      Continuar_M353 : Bool;
      Entrar_M353 : Bool;
      EmiOK_M353 : Bool;
      FinLote_M354 : Bool;
      Especial_M354 : Bool;
      Bit_02_M354 : Bool;
      Retroceder_M354 : Bool;
      Retirar_M354 : Bool;
      Continuar_M354 : Bool;
      Entrar_M354 : Bool;
      EmiOK_M354 : Bool;
      FinLote_M355 : Bool;
      Especial_M355 : Bool;
      Bit_02_M355 : Bool;
      Retroceder_M355 : Bool;
      Retirar_M355 : Bool;
      Continuar_M355 : Bool;
      Entrar_M355 : Bool;
      EmiOK_M355 : Bool;
      FinLote_M356 : Bool;
      Especial_M356 : Bool;
      Bit_02_M356 : Bool;
      Retroceder_M356 : Bool;
      Retirar_M356 : Bool;
      Continuar_M356 : Bool;
      Entrar_M356 : Bool;
      EmiOK_M356 : Bool;
      FinLote_M357 : Bool;
      Especial_M357 : Bool;
      Bit_02_M357 : Bool;
      Retroceder_M357 : Bool;
      Retirar_M357 : Bool;
      Continuar_M357 : Bool;
      Entrar_M357 : Bool;
      EmiOK_M357 : Bool;
      FinLote_M358 : Bool;
      Especial_M358 : Bool;
      Bit_02_M358 : Bool;
      Retroceder_M358 : Bool;
      Retirar_M358 : Bool;
      Continuar_M358 : Bool;
      Entrar_M358 : Bool;
      EmiOK_M358 : Bool;
      FinLote_M359 : Bool;
      Especial_M359 : Bool;
      Bit_02_M359 : Bool;
      Retroceder_M359 : Bool;
      Retirar_M359 : Bool;
      Continuar_M359 : Bool;
      Entrar_M359 : Bool;
      EmiOK_M359 : Bool;
      FinLote_M360 : Bool;
      Especial_M360 : Bool;
      Bit_02_M360 : Bool;
      Retroceder_M360 : Bool;
      Retirar_M360 : Bool;
      Continuar_M360 : Bool;
      Entrar_M360 : Bool;
      EmiOK_M360 : Bool;
      FinLote_M361 : Bool;
      Especial_M361 : Bool;
      Bit_02_M361 : Bool;
      Retroceder_M361 : Bool;
      Retirar_M361 : Bool;
      Continuar_M361 : Bool;
      Entrar_M361 : Bool;
      EmiOK_M361 : Bool;
      FinLote_M362 : Bool;
      Especial_M362 : Bool;
      Bit_02_M362 : Bool;
      Retroceder_M362 : Bool;
      Retirar_M362 : Bool;
      Continuar_M362 : Bool;
      Entrar_M362 : Bool;
      EmiOK_M362 : Bool;
      FinLote_M363 : Bool;
      Especial_M363 : Bool;
      Bit_02_M363 : Bool;
      Retroceder_M363 : Bool;
      Retirar_M363 : Bool;
      Continuar_M363 : Bool;
      Entrar_M363 : Bool;
      EmiOK_M363 : Bool;
      FinLote_M364 : Bool;
      Especial_M364 : Bool;
      Bit_02_M364 : Bool;
      Retroceder_M364 : Bool;
      Retirar_M364 : Bool;
      Continuar_M364 : Bool;
      Entrar_M364 : Bool;
      EmiOK_M364 : Bool;
      FinLote_M365 : Bool;
      Especial_M365 : Bool;
      Bit_02_M365 : Bool;
      Retroceder_M365 : Bool;
      Retirar_M365 : Bool;
      Continuar_M365 : Bool;
      Entrar_M365 : Bool;
      EmiOK_M365 : Bool;
      FinLote_M366 : Bool;
      Especial_M366 : Bool;
      Bit_02_M366 : Bool;
      Retroceder_M366 : Bool;
      Retirar_M366 : Bool;
      Continuar_M366 : Bool;
      Entrar_M366 : Bool;
      EmiOK_M366 : Bool;
      FinLote_M367 : Bool;
      Especial_M367 : Bool;
      Bit_02_M367 : Bool;
      Retroceder_M367 : Bool;
      Retirar_M367 : Bool;
      Continuar_M367 : Bool;
      Entrar_M367 : Bool;
      EmiOK_M367 : Bool;
      FinLote_M368 : Bool;
      Especial_M368 : Bool;
      Bit_02_M368 : Bool;
      Retroceder_M368 : Bool;
      Retirar_M368 : Bool;
      Continuar_M368 : Bool;
      Entrar_M368 : Bool;
      EmiOK_M368 : Bool;
      FinLote_M369 : Bool;
      Especial_M369 : Bool;
      Bit_02_M369 : Bool;
      Retroceder_M369 : Bool;
      Retirar_M369 : Bool;
      Continuar_M369 : Bool;
      Entrar_M369 : Bool;
      EmiOK_M369 : Bool;
      FinLote_M370 : Bool;
      Especial_M370 : Bool;
      Bit_02_M370 : Bool;
      Retroceder_M370 : Bool;
      Retirar_M370 : Bool;
      Continuar_M370 : Bool;
      Entrar_M370 : Bool;
      EmiOK_M370 : Bool;
      FinLote_M371 : Bool;
      Especial_M371 : Bool;
      Bit_02_M371 : Bool;
      Retroceder_M371 : Bool;
      Retirar_M371 : Bool;
      Continuar_M371 : Bool;
      Entrar_M371 : Bool;
      EmiOK_M371 : Bool;
      FinLote_M372 : Bool;
      Especial_M372 : Bool;
      Bit_02_M372 : Bool;
      Retroceder_M372 : Bool;
      Retirar_M372 : Bool;
      Continuar_M372 : Bool;
      Entrar_M372 : Bool;
      EmiOK_M372 : Bool;
      FinLote_M373 : Bool;
      Especial_M373 : Bool;
      Bit_02_M373 : Bool;
      Retroceder_M373 : Bool;
      Retirar_M373 : Bool;
      Continuar_M373 : Bool;
      Entrar_M373 : Bool;
      EmiOK_M373 : Bool;
      FinLote_M374 : Bool;
      Especial_M374 : Bool;
      Bit_02_M374 : Bool;
      Retroceder_M374 : Bool;
      Retirar_M374 : Bool;
      Continuar_M374 : Bool;
      Entrar_M374 : Bool;
      EmiOK_M374 : Bool;
      FinLote_M375 : Bool;
      Especial_M375 : Bool;
      Bit_02_M375 : Bool;
      Retroceder_M375 : Bool;
      Retirar_M375 : Bool;
      Continuar_M375 : Bool;
      Entrar_M375 : Bool;
      EmiOK_M375 : Bool;
      FinLote_M376 : Bool;
      Especial_M376 : Bool;
      Bit_02_M376 : Bool;
      Retroceder_M376 : Bool;
      Retirar_M376 : Bool;
      Continuar_M376 : Bool;
      Entrar_M376 : Bool;
      EmiOK_M376 : Bool;
      FinLote_M377 : Bool;
      Especial_M377 : Bool;
      Bit_02_M377 : Bool;
      Retroceder_M377 : Bool;
      Retirar_M377 : Bool;
      Continuar_M377 : Bool;
      Entrar_M377 : Bool;
      EmiOK_M377 : Bool;
      FinLote_M378 : Bool;
      Especial_M378 : Bool;
      Bit_02_M378 : Bool;
      Retroceder_M378 : Bool;
      Retirar_M378 : Bool;
      Continuar_M378 : Bool;
      Entrar_M378 : Bool;
      EmiOK_M378 : Bool;
      FinLote_M379 : Bool;
      Especial_M379 : Bool;
      Bit_02_M379 : Bool;
      Retroceder_M379 : Bool;
      Retirar_M379 : Bool;
      Continuar_M379 : Bool;
      Entrar_M379 : Bool;
      EmiOK_M379 : Bool;
      FinLote_M380 : Bool;
      Especial_M380 : Bool;
      Bit_02_M380 : Bool;
      Retroceder_M380 : Bool;
      Retirar_M380 : Bool;
      Continuar_M380 : Bool;
      Entrar_M380 : Bool;
      EmiOK_M380 : Bool;
      FinLote_M381 : Bool;
      Especial_M381 : Bool;
      Bit_02_M381 : Bool;
      Retroceder_M381 : Bool;
      Retirar_M381 : Bool;
      Continuar_M381 : Bool;
      Entrar_M381 : Bool;
      EmiOK_M381 : Bool;
      FinLote_M382 : Bool;
      Especial_M382 : Bool;
      Bit_02_M382 : Bool;
      Retroceder_M382 : Bool;
      Retirar_M382 : Bool;
      Continuar_M382 : Bool;
      Entrar_M382 : Bool;
      EmiOK_M382 : Bool;
      FinLote_M383 : Bool;
      Especial_M383 : Bool;
      Bit_02_M383 : Bool;
      Retroceder_M383 : Bool;
      Retirar_M383 : Bool;
      Continuar_M383 : Bool;
      Entrar_M383 : Bool;
      EmiOK_M383 : Bool;
      FinLote_M384 : Bool;
      Especial_M384 : Bool;
      Bit_02_M384 : Bool;
      Retroceder_M384 : Bool;
      Retirar_M384 : Bool;
      Continuar_M384 : Bool;
      Entrar_M384 : Bool;
      EmiOK_M384 : Bool;
      FinLote_M385 : Bool;
      Especial_M385 : Bool;
      Bit_02_M385 : Bool;
      Retroceder_M385 : Bool;
      Retirar_M385 : Bool;
      Continuar_M385 : Bool;
      Entrar_M385 : Bool;
      EmiOK_M385 : Bool;
      FinLote_M386 : Bool;
      Especial_M386 : Bool;
      Bit_02_M386 : Bool;
      Retroceder_M386 : Bool;
      Retirar_M386 : Bool;
      Continuar_M386 : Bool;
      Entrar_M386 : Bool;
      EmiOK_M386 : Bool;
      FinLote_M387 : Bool;
      Especial_M387 : Bool;
      Bit_02_M387 : Bool;
      Retroceder_M387 : Bool;
      Retirar_M387 : Bool;
      Continuar_M387 : Bool;
      Entrar_M387 : Bool;
      EmiOK_M387 : Bool;
      FinLote_M388 : Bool;
      Especial_M388 : Bool;
      Bit_02_M388 : Bool;
      Retroceder_M388 : Bool;
      Retirar_M388 : Bool;
      Continuar_M388 : Bool;
      Entrar_M388 : Bool;
      EmiOK_M388 : Bool;
      FinLote_M389 : Bool;
      Especial_M389 : Bool;
      Bit_02_M389 : Bool;
      Retroceder_M389 : Bool;
      Retirar_M389 : Bool;
      Continuar_M389 : Bool;
      Entrar_M389 : Bool;
      EmiOK_M389 : Bool;
      FinLote_M390 : Bool;
      Especial_M390 : Bool;
      Bit_02_M390 : Bool;
      Retroceder_M390 : Bool;
      Retirar_M390 : Bool;
      Continuar_M390 : Bool;
      Entrar_M390 : Bool;
      EmiOK_M390 : Bool;
      FinLote_M391 : Bool;
      Especial_M391 : Bool;
      Bit_02_M391 : Bool;
      Retroceder_M391 : Bool;
      Retirar_M391 : Bool;
      Continuar_M391 : Bool;
      Entrar_M391 : Bool;
      EmiOK_M391 : Bool;
      FinLote_M392 : Bool;
      Especial_M392 : Bool;
      Bit_02_M392 : Bool;
      Retroceder_M392 : Bool;
      Retirar_M392 : Bool;
      Continuar_M392 : Bool;
      Entrar_M392 : Bool;
      EmiOK_M392 : Bool;
      FinLote_M393 : Bool;
      Especial_M393 : Bool;
      Bit_02_M393 : Bool;
      Retroceder_M393 : Bool;
      Retirar_M393 : Bool;
      Continuar_M393 : Bool;
      Entrar_M393 : Bool;
      EmiOK_M393 : Bool;
      FinLote_M394 : Bool;
      Especial_M394 : Bool;
      Bit_02_M394 : Bool;
      Retroceder_M394 : Bool;
      Retirar_M394 : Bool;
      Continuar_M394 : Bool;
      Entrar_M394 : Bool;
      EmiOK_M394 : Bool;
      FinLote_M395 : Bool;
      Especial_M395 : Bool;
      Bit_02_M395 : Bool;
      Retroceder_M395 : Bool;
      Retirar_M395 : Bool;
      Continuar_M395 : Bool;
      Entrar_M395 : Bool;
      EmiOK_M395 : Bool;
      FinLote_M396 : Bool;
      Especial_M396 : Bool;
      Bit_02_M396 : Bool;
      Retroceder_M396 : Bool;
      Retirar_M396 : Bool;
      Continuar_M396 : Bool;
      Entrar_M396 : Bool;
      EmiOK_M396 : Bool;
      FinLote_M397 : Bool;
      Especial_M397 : Bool;
      Bit_02_M397 : Bool;
      Retroceder_M397 : Bool;
      Retirar_M397 : Bool;
      Continuar_M397 : Bool;
      Entrar_M397 : Bool;
      EmiOK_M397 : Bool;
      FinLote_M398 : Bool;
      Especial_M398 : Bool;
      Bit_02_M398 : Bool;
      Retroceder_M398 : Bool;
      Retirar_M398 : Bool;
      Continuar_M398 : Bool;
      Entrar_M398 : Bool;
      EmiOK_M398 : Bool;
      FinLote_M399 : Bool;
      Especial_M399 : Bool;
      Bit_02_M399 : Bool;
      Retroceder_M399 : Bool;
      Retirar_M399 : Bool;
      Continuar_M399 : Bool;
      Entrar_M399 : Bool;
      EmiOK_M399 : Bool;
      FinLote_M400 : Bool;
      Especial_M400 : Bool;
      Bit_02_M400 : Bool;
      Retroceder_M400 : Bool;
      Retirar_M400 : Bool;
      Continuar_M400 : Bool;
      Entrar_M400 : Bool;
      EmiOK_M400 : Bool;
      FinLote_M401 : Bool;
      Especial_M401 : Bool;
      Bit_02_M401 : Bool;
      Retroceder_M401 : Bool;
      Retirar_M401 : Bool;
      Continuar_M401 : Bool;
      Entrar_M401 : Bool;
      EmiOK_M401 : Bool;
      FinLote_M402 : Bool;
      Especial_M402 : Bool;
      Bit_02_M402 : Bool;
      Retroceder_M402 : Bool;
      Retirar_M402 : Bool;
      Continuar_M402 : Bool;
      Entrar_M402 : Bool;
      EmiOK_M402 : Bool;
      FinLote_M403 : Bool;
      Especial_M403 : Bool;
      Bit_02_M403 : Bool;
      Retroceder_M403 : Bool;
      Retirar_M403 : Bool;
      Continuar_M403 : Bool;
      Entrar_M403 : Bool;
      EmiOK_M403 : Bool;
      FinLote_M404 : Bool;
      Especial_M404 : Bool;
      Bit_02_M404 : Bool;
      Retroceder_M404 : Bool;
      Retirar_M404 : Bool;
      Continuar_M404 : Bool;
      Entrar_M404 : Bool;
      EmiOK_M404 : Bool;
      FinLote_M405 : Bool;
      Especial_M405 : Bool;
      Bit_02_M405 : Bool;
      Retroceder_M405 : Bool;
      Retirar_M405 : Bool;
      Continuar_M405 : Bool;
      Entrar_M405 : Bool;
      EmiOK_M405 : Bool;
      FinLote_M406 : Bool;
      Especial_M406 : Bool;
      Bit_02_M406 : Bool;
      Retroceder_M406 : Bool;
      Retirar_M406 : Bool;
      Continuar_M406 : Bool;
      Entrar_M406 : Bool;
      EmiOK_M406 : Bool;
      FinLote_M407 : Bool;
      Especial_M407 : Bool;
      Bit_02_M407 : Bool;
      Retroceder_M407 : Bool;
      Retirar_M407 : Bool;
      Continuar_M407 : Bool;
      Entrar_M407 : Bool;
      EmiOK_M407 : Bool;
      FinLote_M408 : Bool;
      Especial_M408 : Bool;
      Bit_02_M408 : Bool;
      Retroceder_M408 : Bool;
      Retirar_M408 : Bool;
      Continuar_M408 : Bool;
      Entrar_M408 : Bool;
      EmiOK_M408 : Bool;
      FinLote_M409 : Bool;
      Especial_M409 : Bool;
      Bit_02_M409 : Bool;
      Retroceder_M409 : Bool;
      Retirar_M409 : Bool;
      Continuar_M409 : Bool;
      Entrar_M409 : Bool;
      EmiOK_M409 : Bool;
      FinLote_M410 : Bool;
      Especial_M410 : Bool;
      Bit_02_M410 : Bool;
      Retroceder_M410 : Bool;
      Retirar_M410 : Bool;
      Continuar_M410 : Bool;
      Entrar_M410 : Bool;
      EmiOK_M410 : Bool;
      FinLote_M411 : Bool;
      Especial_M411 : Bool;
      Bit_02_M411 : Bool;
      Retroceder_M411 : Bool;
      Retirar_M411 : Bool;
      Continuar_M411 : Bool;
      Entrar_M411 : Bool;
      EmiOK_M411 : Bool;
      FinLote_M412 : Bool;
      Especial_M412 : Bool;
      Bit_02_M412 : Bool;
      Retroceder_M412 : Bool;
      Retirar_M412 : Bool;
      Continuar_M412 : Bool;
      Entrar_M412 : Bool;
      EmiOK_M412 : Bool;
      FinLote_M413 : Bool;
      Especial_M413 : Bool;
      Bit_02_M413 : Bool;
      Retroceder_M413 : Bool;
      Retirar_M413 : Bool;
      Continuar_M413 : Bool;
      Entrar_M413 : Bool;
      EmiOK_M413 : Bool;
      FinLote_M414 : Bool;
      Especial_M414 : Bool;
      Bit_02_M414 : Bool;
      Retroceder_M414 : Bool;
      Retirar_M414 : Bool;
      Continuar_M414 : Bool;
      Entrar_M414 : Bool;
      EmiOK_M414 : Bool;
      FinLote_M415 : Bool;
      Especial_M415 : Bool;
      Bit_02_M415 : Bool;
      Retroceder_M415 : Bool;
      Retirar_M415 : Bool;
      Continuar_M415 : Bool;
      Entrar_M415 : Bool;
      EmiOK_M415 : Bool;
      FinLote_M416 : Bool;
      Especial_M416 : Bool;
      Bit_02_M416 : Bool;
      Retroceder_M416 : Bool;
      Retirar_M416 : Bool;
      Continuar_M416 : Bool;
      Entrar_M416 : Bool;
      EmiOK_M416 : Bool;
      FinLote_M417 : Bool;
      Especial_M417 : Bool;
      Bit_02_M417 : Bool;
      Retroceder_M417 : Bool;
      Retirar_M417 : Bool;
      Continuar_M417 : Bool;
      Entrar_M417 : Bool;
      EmiOK_M417 : Bool;
      FinLote_M418 : Bool;
      Especial_M418 : Bool;
      Bit_02_M418 : Bool;
      Retroceder_M418 : Bool;
      Retirar_M418 : Bool;
      Continuar_M418 : Bool;
      Entrar_M418 : Bool;
      EmiOK_M418 : Bool;
      FinLote_M419 : Bool;
      Especial_M419 : Bool;
      Bit_02_M419 : Bool;
      Retroceder_M419 : Bool;
      Retirar_M419 : Bool;
      Continuar_M419 : Bool;
      Entrar_M419 : Bool;
      EmiOK_M419 : Bool;
      FinLote_M420 : Bool;
      Especial_M420 : Bool;
      Bit_02_M420 : Bool;
      Retroceder_M420 : Bool;
      Retirar_M420 : Bool;
      Continuar_M420 : Bool;
      Entrar_M420 : Bool;
      EmiOK_M420 : Bool;
      FinLote_M421 : Bool;
      Especial_M421 : Bool;
      Bit_02_M421 : Bool;
      Retroceder_M421 : Bool;
      Retirar_M421 : Bool;
      Continuar_M421 : Bool;
      Entrar_M421 : Bool;
      EmiOK_M421 : Bool;
      FinLote_M422 : Bool;
      Especial_M422 : Bool;
      Bit_02_M422 : Bool;
      Retroceder_M422 : Bool;
      Retirar_M422 : Bool;
      Continuar_M422 : Bool;
      Entrar_M422 : Bool;
      EmiOK_M422 : Bool;
      FinLote_M423 : Bool;
      Especial_M423 : Bool;
      Bit_02_M423 : Bool;
      Retroceder_M423 : Bool;
      Retirar_M423 : Bool;
      Continuar_M423 : Bool;
      Entrar_M423 : Bool;
      EmiOK_M423 : Bool;
      FinLote_M424 : Bool;
      Especial_M424 : Bool;
      Bit_02_M424 : Bool;
      Retroceder_M424 : Bool;
      Retirar_M424 : Bool;
      Continuar_M424 : Bool;
      Entrar_M424 : Bool;
      EmiOK_M424 : Bool;
      FinLote_M425 : Bool;
      Especial_M425 : Bool;
      Bit_02_M425 : Bool;
      Retroceder_M425 : Bool;
      Retirar_M425 : Bool;
      Continuar_M425 : Bool;
      Entrar_M425 : Bool;
      EmiOK_M425 : Bool;
      FinLote_M426 : Bool;
      Especial_M426 : Bool;
      Bit_02_M426 : Bool;
      Retroceder_M426 : Bool;
      Retirar_M426 : Bool;
      Continuar_M426 : Bool;
      Entrar_M426 : Bool;
      EmiOK_M426 : Bool;
      FinLote_M427 : Bool;
      Especial_M427 : Bool;
      Bit_02_M427 : Bool;
      Retroceder_M427 : Bool;
      Retirar_M427 : Bool;
      Continuar_M427 : Bool;
      Entrar_M427 : Bool;
      EmiOK_M427 : Bool;
      FinLote_M428 : Bool;
      Especial_M428 : Bool;
      Bit_02_M428 : Bool;
      Retroceder_M428 : Bool;
      Retirar_M428 : Bool;
      Continuar_M428 : Bool;
      Entrar_M428 : Bool;
      EmiOK_M428 : Bool;
      FinLote_M429 : Bool;
      Especial_M429 : Bool;
      Bit_02_M429 : Bool;
      Retroceder_M429 : Bool;
      Retirar_M429 : Bool;
      Continuar_M429 : Bool;
      Entrar_M429 : Bool;
      EmiOK_M429 : Bool;
      FinLote_M430 : Bool;
      Especial_M430 : Bool;
      Bit_02_M430 : Bool;
      Retroceder_M430 : Bool;
      Retirar_M430 : Bool;
      Continuar_M430 : Bool;
      Entrar_M430 : Bool;
      EmiOK_M430 : Bool;
      FinLote_M431 : Bool;
      Especial_M431 : Bool;
      Bit_02_M431 : Bool;
      Retroceder_M431 : Bool;
      Retirar_M431 : Bool;
      Continuar_M431 : Bool;
      Entrar_M431 : Bool;
      EmiOK_M431 : Bool;
      FinLote_M432 : Bool;
      Especial_M432 : Bool;
      Bit_02_M432 : Bool;
      Retroceder_M432 : Bool;
      Retirar_M432 : Bool;
      Continuar_M432 : Bool;
      Entrar_M432 : Bool;
      EmiOK_M432 : Bool;
      FinLote_M433 : Bool;
      Especial_M433 : Bool;
      Bit_02_M433 : Bool;
      Retroceder_M433 : Bool;
      Retirar_M433 : Bool;
      Continuar_M433 : Bool;
      Entrar_M433 : Bool;
      EmiOK_M433 : Bool;
      FinLote_M434 : Bool;
      Especial_M434 : Bool;
      Bit_02_M434 : Bool;
      Retroceder_M434 : Bool;
      Retirar_M434 : Bool;
      Continuar_M434 : Bool;
      Entrar_M434 : Bool;
      EmiOK_M434 : Bool;
      FinLote_M435 : Bool;
      Especial_M435 : Bool;
      Bit_02_M435 : Bool;
      Retroceder_M435 : Bool;
      Retirar_M435 : Bool;
      Continuar_M435 : Bool;
      Entrar_M435 : Bool;
      EmiOK_M435 : Bool;
      FinLote_M436 : Bool;
      Especial_M436 : Bool;
      Bit_02_M436 : Bool;
      Retroceder_M436 : Bool;
      Retirar_M436 : Bool;
      Continuar_M436 : Bool;
      Entrar_M436 : Bool;
      EmiOK_M436 : Bool;
      FinLote_M437 : Bool;
      Especial_M437 : Bool;
      Bit_02_M437 : Bool;
      Retroceder_M437 : Bool;
      Retirar_M437 : Bool;
      Continuar_M437 : Bool;
      Entrar_M437 : Bool;
      EmiOK_M437 : Bool;
      FinLote_M438 : Bool;
      Especial_M438 : Bool;
      Bit_02_M438 : Bool;
      Retroceder_M438 : Bool;
      Retirar_M438 : Bool;
      Continuar_M438 : Bool;
      Entrar_M438 : Bool;
      EmiOK_M438 : Bool;
      FinLote_M439 : Bool;
      Especial_M439 : Bool;
      Bit_02_M439 : Bool;
      Retroceder_M439 : Bool;
      Retirar_M439 : Bool;
      Continuar_M439 : Bool;
      Entrar_M439 : Bool;
      EmiOK_M439 : Bool;
      FinLote_M440 : Bool;
      Especial_M440 : Bool;
      Bit_02_M440 : Bool;
      Retroceder_M440 : Bool;
      Retirar_M440 : Bool;
      Continuar_M440 : Bool;
      Entrar_M440 : Bool;
      EmiOK_M440 : Bool;
      FinLote_M441 : Bool;
      Especial_M441 : Bool;
      Bit_02_M441 : Bool;
      Retroceder_M441 : Bool;
      Retirar_M441 : Bool;
      Continuar_M441 : Bool;
      Entrar_M441 : Bool;
      EmiOK_M441 : Bool;
      FinLote_M442 : Bool;
      Especial_M442 : Bool;
      Bit_02_M442 : Bool;
      Retroceder_M442 : Bool;
      Retirar_M442 : Bool;
      Continuar_M442 : Bool;
      Entrar_M442 : Bool;
      EmiOK_M442 : Bool;
      FinLote_M443 : Bool;
      Especial_M443 : Bool;
      Bit_02_M443 : Bool;
      Retroceder_M443 : Bool;
      Retirar_M443 : Bool;
      Continuar_M443 : Bool;
      Entrar_M443 : Bool;
      EmiOK_M443 : Bool;
      FinLote_M444 : Bool;
      Especial_M444 : Bool;
      Bit_02_M444 : Bool;
      Retroceder_M444 : Bool;
      Retirar_M444 : Bool;
      Continuar_M444 : Bool;
      Entrar_M444 : Bool;
      EmiOK_M444 : Bool;
      FinLote_M445 : Bool;
      Especial_M445 : Bool;
      Bit_02_M445 : Bool;
      Retroceder_M445 : Bool;
      Retirar_M445 : Bool;
      Continuar_M445 : Bool;
      Entrar_M445 : Bool;
      EmiOK_M445 : Bool;
      FinLote_M446 : Bool;
      Especial_M446 : Bool;
      Bit_02_M446 : Bool;
      Retroceder_M446 : Bool;
      Retirar_M446 : Bool;
      Continuar_M446 : Bool;
      Entrar_M446 : Bool;
      EmiOK_M446 : Bool;
      FinLote_M447 : Bool;
      Especial_M447 : Bool;
      Bit_02_M447 : Bool;
      Retroceder_M447 : Bool;
      Retirar_M447 : Bool;
      Continuar_M447 : Bool;
      Entrar_M447 : Bool;
      EmiOK_M447 : Bool;
      FinLote_M448 : Bool;
      Especial_M448 : Bool;
      Bit_02_M448 : Bool;
      Retroceder_M448 : Bool;
      Retirar_M448 : Bool;
      Continuar_M448 : Bool;
      Entrar_M448 : Bool;
      EmiOK_M448 : Bool;
      FinLote_M449 : Bool;
      Especial_M449 : Bool;
      Bit_02_M449 : Bool;
      Retroceder_M449 : Bool;
      Retirar_M449 : Bool;
      Continuar_M449 : Bool;
      Entrar_M449 : Bool;
      EmiOK_M449 : Bool;
      FinLote_M450 : Bool;
      Especial_M450 : Bool;
      Bit_02_M450 : Bool;
      Retroceder_M450 : Bool;
      Retirar_M450 : Bool;
      Continuar_M450 : Bool;
      Entrar_M450 : Bool;
      EmiOK_M450 : Bool;
      FinLote_M451 : Bool;
      Especial_M451 : Bool;
      Bit_02_M451 : Bool;
      Retroceder_M451 : Bool;
      Retirar_M451 : Bool;
      Continuar_M451 : Bool;
      Entrar_M451 : Bool;
      EmiOK_M451 : Bool;
      FinLote_M452 : Bool;
      Especial_M452 : Bool;
      Bit_02_M452 : Bool;
      Retroceder_M452 : Bool;
      Retirar_M452 : Bool;
      Continuar_M452 : Bool;
      Entrar_M452 : Bool;
      EmiOK_M452 : Bool;
      FinLote_M453 : Bool;
      Especial_M453 : Bool;
      Bit_02_M453 : Bool;
      Retroceder_M453 : Bool;
      Retirar_M453 : Bool;
      Continuar_M453 : Bool;
      Entrar_M453 : Bool;
      EmiOK_M453 : Bool;
      FinLote_M454 : Bool;
      Especial_M454 : Bool;
      Bit_02_M454 : Bool;
      Retroceder_M454 : Bool;
      Retirar_M454 : Bool;
      Continuar_M454 : Bool;
      Entrar_M454 : Bool;
      EmiOK_M454 : Bool;
      FinLote_M455 : Bool;
      Especial_M455 : Bool;
      Bit_02_M455 : Bool;
      Retroceder_M455 : Bool;
      Retirar_M455 : Bool;
      Continuar_M455 : Bool;
      Entrar_M455 : Bool;
      EmiOK_M455 : Bool;
      FinLote_M456 : Bool;
      Especial_M456 : Bool;
      Bit_02_M456 : Bool;
      Retroceder_M456 : Bool;
      Retirar_M456 : Bool;
      Continuar_M456 : Bool;
      Entrar_M456 : Bool;
      EmiOK_M456 : Bool;
      FinLote_M457 : Bool;
      Especial_M457 : Bool;
      Bit_02_M457 : Bool;
      Retroceder_M457 : Bool;
      Retirar_M457 : Bool;
      Continuar_M457 : Bool;
      Entrar_M457 : Bool;
      EmiOK_M457 : Bool;
      FinLote_M458 : Bool;
      Especial_M458 : Bool;
      Bit_02_M458 : Bool;
      Retroceder_M458 : Bool;
      Retirar_M458 : Bool;
      Continuar_M458 : Bool;
      Entrar_M458 : Bool;
      EmiOK_M458 : Bool;
      FinLote_M459 : Bool;
      Especial_M459 : Bool;
      Bit_02_M459 : Bool;
      Retroceder_M459 : Bool;
      Retirar_M459 : Bool;
      Continuar_M459 : Bool;
      Entrar_M459 : Bool;
      EmiOK_M459 : Bool;
      FinLote_M460 : Bool;
      Especial_M460 : Bool;
      Bit_02_M460 : Bool;
      Retroceder_M460 : Bool;
      Retirar_M460 : Bool;
      Continuar_M460 : Bool;
      Entrar_M460 : Bool;
      EmiOK_M460 : Bool;
      FinLote_M461 : Bool;
      Especial_M461 : Bool;
      Bit_02_M461 : Bool;
      Retroceder_M461 : Bool;
      Retirar_M461 : Bool;
      Continuar_M461 : Bool;
      Entrar_M461 : Bool;
      EmiOK_M461 : Bool;
      FinLote_M462 : Bool;
      Especial_M462 : Bool;
      Bit_02_M462 : Bool;
      Retroceder_M462 : Bool;
      Retirar_M462 : Bool;
      Continuar_M462 : Bool;
      Entrar_M462 : Bool;
      EmiOK_M462 : Bool;
      FinLote_M463 : Bool;
      Especial_M463 : Bool;
      Bit_02_M463 : Bool;
      Retroceder_M463 : Bool;
      Retirar_M463 : Bool;
      Continuar_M463 : Bool;
      Entrar_M463 : Bool;
      EmiOK_M463 : Bool;
      FinLote_M464 : Bool;
      Especial_M464 : Bool;
      Bit_02_M464 : Bool;
      Retroceder_M464 : Bool;
      Retirar_M464 : Bool;
      Continuar_M464 : Bool;
      Entrar_M464 : Bool;
      EmiOK_M464 : Bool;
      FinLote_M465 : Bool;
      Especial_M465 : Bool;
      Bit_02_M465 : Bool;
      Retroceder_M465 : Bool;
      Retirar_M465 : Bool;
      Continuar_M465 : Bool;
      Entrar_M465 : Bool;
      EmiOK_M465 : Bool;
      FinLote_M466 : Bool;
      Especial_M466 : Bool;
      Bit_02_M466 : Bool;
      Retroceder_M466 : Bool;
      Retirar_M466 : Bool;
      Continuar_M466 : Bool;
      Entrar_M466 : Bool;
      EmiOK_M466 : Bool;
      FinLote_M467 : Bool;
      Especial_M467 : Bool;
      Bit_02_M467 : Bool;
      Retroceder_M467 : Bool;
      Retirar_M467 : Bool;
      Continuar_M467 : Bool;
      Entrar_M467 : Bool;
      EmiOK_M467 : Bool;
      FinLote_M468 : Bool;
      Especial_M468 : Bool;
      Bit_02_M468 : Bool;
      Retroceder_M468 : Bool;
      Retirar_M468 : Bool;
      Continuar_M468 : Bool;
      Entrar_M468 : Bool;
      EmiOK_M468 : Bool;
      FinLote_M469 : Bool;
      Especial_M469 : Bool;
      Bit_02_M469 : Bool;
      Retroceder_M469 : Bool;
      Retirar_M469 : Bool;
      Continuar_M469 : Bool;
      Entrar_M469 : Bool;
      EmiOK_M469 : Bool;
      FinLote_M470 : Bool;
      Especial_M470 : Bool;
      Bit_02_M470 : Bool;
      Retroceder_M470 : Bool;
      Retirar_M470 : Bool;
      Continuar_M470 : Bool;
      Entrar_M470 : Bool;
      EmiOK_M470 : Bool;
      FinLote_M471 : Bool;
      Especial_M471 : Bool;
      Bit_02_M471 : Bool;
      Retroceder_M471 : Bool;
      Retirar_M471 : Bool;
      Continuar_M471 : Bool;
      Entrar_M471 : Bool;
      EmiOK_M471 : Bool;
      FinLote_M472 : Bool;
      Especial_M472 : Bool;
      Bit_02_M472 : Bool;
      Retroceder_M472 : Bool;
      Retirar_M472 : Bool;
      Continuar_M472 : Bool;
      Entrar_M472 : Bool;
      EmiOK_M472 : Bool;
      FinLote_M473 : Bool;
      Especial_M473 : Bool;
      Bit_02_M473 : Bool;
      Retroceder_M473 : Bool;
      Retirar_M473 : Bool;
      Continuar_M473 : Bool;
      Entrar_M473 : Bool;
      EmiOK_M473 : Bool;
      FinLote_M474 : Bool;
      Especial_M474 : Bool;
      Bit_02_M474 : Bool;
      Retroceder_M474 : Bool;
      Retirar_M474 : Bool;
      Continuar_M474 : Bool;
      Entrar_M474 : Bool;
      EmiOK_M474 : Bool;
      FinLote_M475 : Bool;
      Especial_M475 : Bool;
      Bit_02_M475 : Bool;
      Retroceder_M475 : Bool;
      Retirar_M475 : Bool;
      Continuar_M475 : Bool;
      Entrar_M475 : Bool;
      EmiOK_M475 : Bool;
      FinLote_M476 : Bool;
      Especial_M476 : Bool;
      Bit_02_M476 : Bool;
      Retroceder_M476 : Bool;
      Retirar_M476 : Bool;
      Continuar_M476 : Bool;
      Entrar_M476 : Bool;
      EmiOK_M476 : Bool;
      FinLote_M477 : Bool;
      Especial_M477 : Bool;
      Bit_02_M477 : Bool;
      Retroceder_M477 : Bool;
      Retirar_M477 : Bool;
      Continuar_M477 : Bool;
      Entrar_M477 : Bool;
      EmiOK_M477 : Bool;
      FinLote_M478 : Bool;
      Especial_M478 : Bool;
      Bit_02_M478 : Bool;
      Retroceder_M478 : Bool;
      Retirar_M478 : Bool;
      Continuar_M478 : Bool;
      Entrar_M478 : Bool;
      EmiOK_M478 : Bool;
      FinLote_M479 : Bool;
      Especial_M479 : Bool;
      Bit_02_M479 : Bool;
      Retroceder_M479 : Bool;
      Retirar_M479 : Bool;
      Continuar_M479 : Bool;
      Entrar_M479 : Bool;
      EmiOK_M479 : Bool;
      FinLote_M480 : Bool;
      Especial_M480 : Bool;
      Bit_02_M480 : Bool;
      Retroceder_M480 : Bool;
      Retirar_M480 : Bool;
      Continuar_M480 : Bool;
      Entrar_M480 : Bool;
      EmiOK_M480 : Bool;
      FinLote_M481 : Bool;
      Especial_M481 : Bool;
      Bit_02_M481 : Bool;
      Retroceder_M481 : Bool;
      Retirar_M481 : Bool;
      Continuar_M481 : Bool;
      Entrar_M481 : Bool;
      EmiOK_M481 : Bool;
      FinLote_M482 : Bool;
      Especial_M482 : Bool;
      Bit_02_M482 : Bool;
      Retroceder_M482 : Bool;
      Retirar_M482 : Bool;
      Continuar_M482 : Bool;
      Entrar_M482 : Bool;
      EmiOK_M482 : Bool;
      FinLote_M483 : Bool;
      Especial_M483 : Bool;
      Bit_02_M483 : Bool;
      Retroceder_M483 : Bool;
      Retirar_M483 : Bool;
      Continuar_M483 : Bool;
      Entrar_M483 : Bool;
      EmiOK_M483 : Bool;
      FinLote_M484 : Bool;
      Especial_M484 : Bool;
      Bit_02_M484 : Bool;
      Retroceder_M484 : Bool;
      Retirar_M484 : Bool;
      Continuar_M484 : Bool;
      Entrar_M484 : Bool;
      EmiOK_M484 : Bool;
      FinLote_M485 : Bool;
      Especial_M485 : Bool;
      Bit_02_M485 : Bool;
      Retroceder_M485 : Bool;
      Retirar_M485 : Bool;
      Continuar_M485 : Bool;
      Entrar_M485 : Bool;
      EmiOK_M485 : Bool;
      FinLote_M486 : Bool;
      Especial_M486 : Bool;
      Bit_02_M486 : Bool;
      Retroceder_M486 : Bool;
      Retirar_M486 : Bool;
      Continuar_M486 : Bool;
      Entrar_M486 : Bool;
      EmiOK_M486 : Bool;
      FinLote_M487 : Bool;
      Especial_M487 : Bool;
      Bit_02_M487 : Bool;
      Retroceder_M487 : Bool;
      Retirar_M487 : Bool;
      Continuar_M487 : Bool;
      Entrar_M487 : Bool;
      EmiOK_M487 : Bool;
      FinLote_M488 : Bool;
      Especial_M488 : Bool;
      Bit_02_M488 : Bool;
      Retroceder_M488 : Bool;
      Retirar_M488 : Bool;
      Continuar_M488 : Bool;
      Entrar_M488 : Bool;
      EmiOK_M488 : Bool;
      FinLote_M489 : Bool;
      Especial_M489 : Bool;
      Bit_02_M489 : Bool;
      Retroceder_M489 : Bool;
      Retirar_M489 : Bool;
      Continuar_M489 : Bool;
      Entrar_M489 : Bool;
      EmiOK_M489 : Bool;
      FinLote_M490 : Bool;
      Especial_M490 : Bool;
      Bit_02_M490 : Bool;
      Retroceder_M490 : Bool;
      Retirar_M490 : Bool;
      Continuar_M490 : Bool;
      Entrar_M490 : Bool;
      EmiOK_M490 : Bool;
      FinLote_M491 : Bool;
      Especial_M491 : Bool;
      Bit_02_M491 : Bool;
      Retroceder_M491 : Bool;
      Retirar_M491 : Bool;
      Continuar_M491 : Bool;
      Entrar_M491 : Bool;
      EmiOK_M491 : Bool;
      FinLote_M492 : Bool;
      Especial_M492 : Bool;
      Bit_02_M492 : Bool;
      Retroceder_M492 : Bool;
      Retirar_M492 : Bool;
      Continuar_M492 : Bool;
      Entrar_M492 : Bool;
      EmiOK_M492 : Bool;
      FinLote_M493 : Bool;
      Especial_M493 : Bool;
      Bit_02_M493 : Bool;
      Retroceder_M493 : Bool;
      Retirar_M493 : Bool;
      Continuar_M493 : Bool;
      Entrar_M493 : Bool;
      EmiOK_M493 : Bool;
      FinLote_M494 : Bool;
      Especial_M494 : Bool;
      Bit_02_M494 : Bool;
      Retroceder_M494 : Bool;
      Retirar_M494 : Bool;
      Continuar_M494 : Bool;
      Entrar_M494 : Bool;
      EmiOK_M494 : Bool;
      FinLote_M495 : Bool;
      Especial_M495 : Bool;
      Bit_02_M495 : Bool;
      Retroceder_M495 : Bool;
      Retirar_M495 : Bool;
      Continuar_M495 : Bool;
      Entrar_M495 : Bool;
      EmiOK_M495 : Bool;
      FinLote_M496 : Bool;
      Especial_M496 : Bool;
      Bit_02_M496 : Bool;
      Retroceder_M496 : Bool;
      Retirar_M496 : Bool;
      Continuar_M496 : Bool;
      Entrar_M496 : Bool;
      EmiOK_M496 : Bool;
      FinLote_M497 : Bool;
      Especial_M497 : Bool;
      Bit_02_M497 : Bool;
      Retroceder_M497 : Bool;
      Retirar_M497 : Bool;
      Continuar_M497 : Bool;
      Entrar_M497 : Bool;
      EmiOK_M497 : Bool;
      FinLote_M498 : Bool;
      Especial_M498 : Bool;
      Bit_02_M498 : Bool;
      Retroceder_M498 : Bool;
      Retirar_M498 : Bool;
      Continuar_M498 : Bool;
      Entrar_M498 : Bool;
      EmiOK_M498 : Bool;
      FinLote_M499 : Bool;
      Especial_M499 : Bool;
      Bit_02_M499 : Bool;
      Retroceder_M499 : Bool;
      Retirar_M499 : Bool;
      Continuar_M499 : Bool;
      Entrar_M499 : Bool;
      EmiOK_M499 : Bool;
      FinLote_M500 : Bool;
      Especial_M500 : Bool;
      Bit_02_M500 : Bool;
      Retroceder_M500 : Bool;
      Retirar_M500 : Bool;
      Continuar_M500 : Bool;
      Entrar_M500 : Bool;
      EmiOK_M500 : Bool;
      Bit_00_CCPIF : Bool;
      Bit_01_CCPIF : Bool;
      Rearme_CCPIF : Bool;
      Bit_03_CCPIF : Bool;
      Reset_CCPIF : Bool;
      Paro_CCPIF : Bool;
      Marcha_CCPIF : Bool;
      EmiOK_CCPIF : Bool;
      Bit_00_CBOX1 : Bool;
      Bit_01_CBOX1 : Bool;
      Rearme_CBOX1 : Bool;
      Bit_03_CBOX1 : Bool;
      Reset_CBOX1 : Bool;
      Paro_CBOX1 : Bool;
      Marcha_CBOX1 : Bool;
      EmiOK_CBOX1 : Bool;
      Bit_00_CBOX2 : Bool;
      Bit_01_CBOX2 : Bool;
      Rearme_CBOX2 : Bool;
      Bit_03_CBOX2 : Bool;
      Reset_CBOX2 : Bool;
      Paro_CBOX2 : Bool;
      Marcha_CBOX2 : Bool;
      EmiOK_CBOX2 : Bool;
      Bit_00_CBOX3 : Bool;
      Bit_01_CBOX3 : Bool;
      Rearme_CBOX3 : Bool;
      Bit_03_CBOX3 : Bool;
      Reset_CBOX3 : Bool;
      Paro_CBOX3 : Bool;
      Marcha_CBOX3 : Bool;
      EmiOK_CBOX3 : Bool;
      Bit_00_CBOX4 : Bool;
      Bit_01_CBOX4 : Bool;
      Rearme_CBOX4 : Bool;
      Bit_03_CBOX4 : Bool;
      Reset_CBOX4 : Bool;
      Paro_CBOX4 : Bool;
      Marcha_CBOX4 : Bool;
      EmiOK_CBOX4 : Bool;
      Bit_00_CBOX5 : Bool;
      Bit_01_CBOX5 : Bool;
      Rearme_CBOX5 : Bool;
      Bit_03_CBOX5 : Bool;
      Reset_CBOX5 : Bool;
      Paro_CBOX5 : Bool;
      Marcha_CBOX5 : Bool;
      EmiOK_CBOX5 : Bool;
      Bit_00_CBOX6 : Bool;
      Bit_01_CBOX6 : Bool;
      Rearme_CBOX6 : Bool;
      Bit_03_CBOX6 : Bool;
      Reset_CBOX6 : Bool;
      Paro_CBOX6 : Bool;
      Marcha_CBOX6 : Bool;
      EmiOK_CBOX6 : Bool;
      Bit_00_CBOX7 : Bool;
      Bit_01_CBOX7 : Bool;
      Rearme_CBOX7 : Bool;
      Bit_03_CBOX7 : Bool;
      Reset_CBOX7 : Bool;
      Paro_CBOX7 : Bool;
      Marcha_CBOX7 : Bool;
      EmiOK_CBOX7 : Bool;
      Bit_00_CBOX8 : Bool;
      Bit_01_CBOX8 : Bool;
      Rearme_CBOX8 : Bool;
      Bit_03_CBOX8 : Bool;
      Reset_CBOX8 : Bool;
      Paro_CBOX8 : Bool;
      Marcha_CBOX8 : Bool;
      EmiOK_CBOX8 : Bool;
      Bit_00_CBOX9 : Bool;
      Bit_01_CBOX9 : Bool;
      Rearme_CBOX9 : Bool;
      Bit_03_CBOX9 : Bool;
      Reset_CBOX9 : Bool;
      Paro_CBOX9 : Bool;
      Marcha_CBOX9 : Bool;
      EmiOK_CBOX9 : Bool;
      Especial : Array[1..128] of Word;
   END_VAR
BEGIN
END_DATA_BLOCK

DATA_BLOCK "DB601_PeinesQuimarox"   // DB601
{ S7_Optimized_Access := 'FALSE' }
AUTHOR : Naibes
// stored: AutoNumber false
   VAR RETAIN
      Quimarox : Array[1.."CTE_MaxNumQuimarox"] of Struct
         vagon { S7_SetPoint := 'True'} : Array[1.."CTE_MaxNumVagones"] of "CBS_Carrier";
      END_STRUCT;
   END_VAR
BEGIN
END_DATA_BLOCK

DATA_BLOCK "DB602_ElementosQuimarox"   // DB602
{ S7_Optimized_Access := 'FALSE' }
// stored: AutoNumber false
   VAR RETAIN
      Quimarox : Array[1.."CTE_MaxNumQuimarox"] of Struct
         Elementos { S7_SetPoint := 'True'} : Array[1.."CTE_MaxNumElementos"] of "CBS_Elemento";
      END_STRUCT;
   END_VAR
BEGIN
   Quimarox[1].Elementos[1].posicion_real_elemento := 700.0;
   Quimarox[1].Elementos[2].posicion_real_elemento := 7700.0;
   Quimarox[1].Elementos[3].posicion_real_elemento := 14890.0;
   Quimarox[1].Elementos[4].posicion_real_elemento := 18000.0;
   Quimarox[1].Elementos[5].posicion_real_elemento := 6870.7;
   Quimarox[1].Elementos[1..5].ventana_minima := 50;
   Quimarox[1].Elementos[1].ventana_maxima := 1400;
   Quimarox[1].Elementos[2..5].ventana_maxima := 1550;
   Quimarox[1].Elementos[6..50].Numero_carrier := 11;
   Quimarox[1].Elementos[6..34].Avance_carrier := 1069;
   Quimarox[1].Elementos[35..47].Avance_carrier := 1079;
   Quimarox[1].Elementos[48..50].Avance_carrier := 1083;
END_DATA_BLOCK

DATA_BLOCK "DB1903_ASI_DIAG"   // DB1903
{ S7_Optimized_Access := 'FALSE'; DB_Accessible_From_OPC_UA := 'FALSE' }
// stored: AutoNumber false, DBAccessibleFromOPCUA false
   VAR
      ASI_Gateway_Error : Bool;
      IP_GW { S7_SetPoint := 'True'} : Array[1..16] of "ASI_GW_DATOS";
      ASI3_GW_C1 : Array[1..16] of "ASI3_Diag_GW";
      ASI3_GW_C2 : Array[1..16] of "ASI3_Diag_GW";
      ASI5_GW_Flags { S7_SetPoint := 'True'} : Array[1..16] of "ASI5_Flags";
      ASI5_GW_C1 : Array[1..16] of "ASI5_Diag_GW";
      ASI5_GW_C2 : Array[1..16] of "ASI5_Diag_GW";
   END_VAR
BEGIN
END_DATA_BLOCK

ORGANIZATION_BLOCK "OB1_Principal"   // OB1, LAD, ProgramCycle
TITLE = "Main Program Sweep (Cycle)"
{ S7_Optimized_Access := 'FALSE' }
AUTHOR : ESTANDAR
NAME : 20150525
VERSION : 3.1
// stored: AutoNumber false, SetENOAutomatically false
   VAR_TEMP
      OB1_EV_CLASS : Byte;   // Bits 0-3 = 1 (Coming event), Bits 4-7 = 1 (Event class 1)
      OB1_SCAN_1 : Byte;   // 1 (Cold restart scan 1 of OB 1), 3 (Scan 2-n of OB 1)
      OB1_PRIORITY : Byte;   // Priority of OB Execution
      OB1_OB_NUMBR : Byte;   // 1 (Organization block 1, OB1)
      OB1_RESERVED_1 : Byte;   // Reserved for system
      OB1_RESERVED_2 : Byte;   // Reserved for system
      OB1_PREV_CYCLE : Int;   // Cycle time of previous OB1 scan (milliseconds)
      OB1_MIN_CYCLE : Int;   // Minimum cycle time of OB1 (milliseconds)
      OB1_MAX_CYCLE : Int;   // Maximum cycle time of OB1 (milliseconds)
      OB1_DATE_TIME : Date_And_Time;   // Date and time OB1 started
      indice : UInt;
   END_VAR
   VAR_TEMP   // added for the SCL form of the ladder/FBD networks
      _w1 : Bool;
   END_VAR
BEGIN

REGION Network 1: Marcas Auxiliares CCPIF
   // *******************************************************************
   // * FUNCION: Generación marcas Auxiliares Generales del sistema     *
   // *******************************************************************
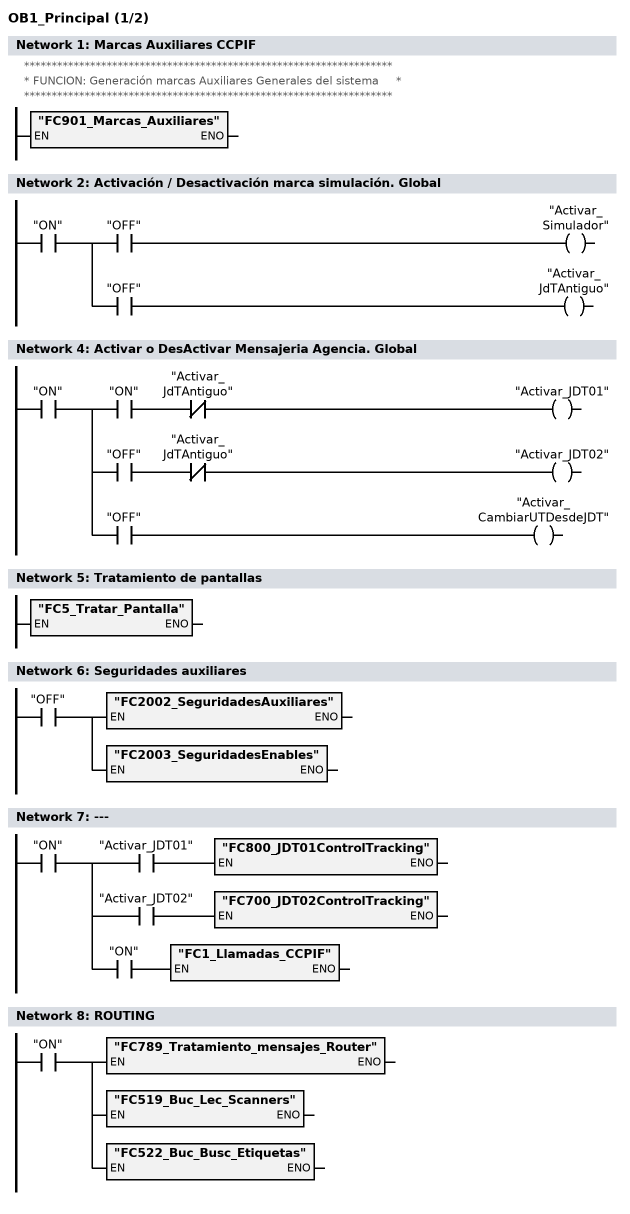
   RUNG wire#powerrail
      "FC901_Marcas_Auxiliares"()
   END_RUNG
   // the same network as SCL:
   "FC901_Marcas_Auxiliares"();
END_REGION

REGION Network 2: Activación / Desactivación marca simulación. Global
   RUNG wire#powerrail
      Contact( "ON" )
      wire#w1
      Contact( "OFF" )
      Coil( "Activar_Simulador" )
   END_RUNG
   RUNG wire#w1
      Contact( "OFF" )
      Coil( "Activar_JdTAntiguo" )
   END_RUNG
   // the same network as SCL:
   "Activar_Simulador" := "ON" AND "OFF";
   "Activar_JdTAntiguo" := "ON" AND "OFF";
END_REGION

NETWORK
TITLE = Cuando se desactive el JDT antiguo, tenemos que borrarnos todas las ordenes que se pudiesen quedar activas
// de lo contrario, habria problemas al realizar el cambio. Pablo
////////////////////////////////////////////////////////////////////////
////////////////////////////////////////////////////////////////////////
////////////////////////////////////////////////////////////////////////
/// --- Control de Cambio de Modo
      SET;
      A     "Activar_JdTAntiguo";
      FN    "Memo_JdTAntiguo_Desactivado";
      JC    BorradoDatos_CambioModo;

      SET;
      A     "Activar_JdTAntiguo";
      FP    "Memo_JdTAntiguo_Activado";
      JC    BorradoDatos_CambioModo;

      JU    Fin_CambioModo;

////////////////////////////////////////////////////////////////////////
////////////////////////////////////////////////////////////////////////
////////////////////////////////////////////////////////////////////////
/// --- Borrado de Datos
BorradoDatos_CambioModo:NOP   0;
      SET;
      S     "DB801_JDT01StatusCOM".ResetBD;
      S     "DB701_JDT02StatusCOM".ResetBD;


////////////////////////////////////////////////////////////////////////
////////////////////////////////////////////////////////////////////////
////////////////////////////////////////////////////////////////////////
/// --- Final de Cambio de Modo
Fin_CambioModo:NOP   0;



REGION Network 4: Activar o DesActivar Mensajeria Agencia. Global
   RUNG wire#powerrail
      Contact( "ON" )
      wire#w1
      Contact( "ON" )
      I_Contact( "Activar_JdTAntiguo" )
      Coil( "Activar_JDT01" )
   END_RUNG
   RUNG wire#w1
      Contact( "OFF" )
      I_Contact( "Activar_JdTAntiguo" )
      Coil( "Activar_JDT02" )
   END_RUNG
   RUNG wire#w1
      Contact( "OFF" )
      Coil( "Activar_CambiarUTDesdeJDT" )
   END_RUNG
   // the same network as SCL:
   "Activar_JDT01" := "ON" AND "ON" AND NOT "Activar_JdTAntiguo";
   "Activar_JDT02" := "ON" AND "OFF" AND NOT "Activar_JdTAntiguo";
   "Activar_CambiarUTDesdeJDT" := "ON" AND "OFF";
END_REGION

REGION Network 5: Tratamiento de pantallas
   RUNG wire#powerrail
      "FC5_Tratar_Pantalla"()
   END_RUNG
   // the same network as SCL:
   "FC5_Tratar_Pantalla"();
END_REGION

REGION Network 6: Seguridades auxiliares
   RUNG wire#powerrail
      Contact( "OFF" )
      wire#w1
      "FC2002_SeguridadesAuxiliares"()
   END_RUNG
   RUNG wire#w1
      "FC2003_SeguridadesEnables"()
   END_RUNG
   // the same network as SCL:
   #_w1 := "OFF";
   IF #_w1 THEN
       "FC2002_SeguridadesAuxiliares"();
       "FC2003_SeguridadesEnables"();
   END_IF;
END_REGION

REGION Network 7: ---
   RUNG wire#powerrail
      Contact( "ON" )
      wire#w1
      Contact( "Activar_JDT01" )
      "FC800_JDT01ControlTracking"()
   END_RUNG
   RUNG wire#w1
      Contact( "Activar_JDT02" )
      "FC700_JDT02ControlTracking"()
   END_RUNG
   RUNG wire#w1
      Contact( "ON" )
      "FC1_Llamadas_CCPIF"()
   END_RUNG
   // the same network as SCL:
   #_w1 := "ON";
   IF "ON" AND "Activar_JDT01" THEN "FC800_JDT01ControlTracking"(); END_IF;
   IF #_w1 AND "Activar_JDT02" THEN "FC700_JDT02ControlTracking"(); END_IF;
   IF #_w1 AND "ON" THEN "FC1_Llamadas_CCPIF"(); END_IF;
END_REGION

REGION Network 8: ROUTING
   RUNG wire#powerrail
      Contact( "ON" )
      wire#w1
      "FC789_Tratamiento_mensajes_Router"()
   END_RUNG
   RUNG wire#w1
      "FC519_Buc_Lec_Scanners"()
   END_RUNG
   RUNG wire#w1
      "FC522_Buc_Busc_Etiquetas"()
   END_RUNG
   // the same network as SCL:
   #_w1 := "ON";
   IF #_w1 THEN
       "FC789_Tratamiento_mensajes_Router"();
       "FC519_Buc_Lec_Scanners"();
       "FC522_Buc_Busc_Etiquetas"();
   END_IF;
END_REGION

REGION Network 9: Llamadas CBOXES
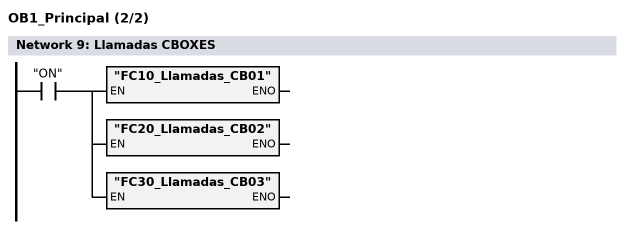
   RUNG wire#powerrail
      Contact( "ON" )
      wire#w1
      "FC10_Llamadas_CB01"()
   END_RUNG
   RUNG wire#w1
      "FC20_Llamadas_CB02"()
   END_RUNG
   RUNG wire#w1
      "FC30_Llamadas_CB03"()
   END_RUNG
   // the same network as SCL:
   #_w1 := "ON";
   IF #_w1 THEN
       "FC10_Llamadas_CB01"();
       "FC20_Llamadas_CB02"();
       "FC30_Llamadas_CB03"();
   END_IF;
END_REGION

NETWORK
TITLE = Configuracion de Mesas >> Activar JDT Antiguo
///////////////////////////////////////////////////////////////////////////
///////////////////////////////////////////////////////////////////////////
///////////////////////////////////////////////////////////////////////////
/// Configuracion de Mesas >> Activar JDT Antiguo
      SET;
      AN    "Activar_JdTAntiguo";
      JC    FinalConfigMesas;


///////////////////////////////////////////////////////////////////////////
/// DeActivar Error De Datos
      L     1;
      T     #indice;

InicioBucle_ConfigMesas:NOP   0;
      SET;
      =     "DB850_DefinicionMesas".Mesa[#indice].ConfigMesa.SinErrorDeDatosCargada;
      =     "DB850_DefinicionMesas".Mesa[#indice].ConfigMesa.SinErrorDeDatosVacia;

      L     #indice;
      L     1;
      +I;
      T     #indice;

      L     #indice;
      L     "CTE_MaxMesas";
      >I;
      JC    FinalConfigMesas;
      JU    InicioBucle_ConfigMesas;


///////////////////////////////////////////////////////////////////////////
///////////////////////////////////////////////////////////////////////////
///////////////////////////////////////////////////////////////////////////
/// Final de Configuracion de Mesas >> Activar JDT Antiguo
FinalConfigMesas:NOP   0;


END_ORGANIZATION_BLOCK

FUNCTION "FC901_Marcas_Auxiliares" : Void   // FC901, LAD
{ S7_Optimized_Access := 'FALSE' }
AUTHOR : GENERAL
NAME : 20130301
VERSION : 3.0
// stored: AutoNumber false, SetENOAutomatically false
   VAR_TEMP
      Incremento_Tiempo : Time;
      Aux_Ret_Val : Int;
      Fecha_Actual : Date;
      Hora : Time_Of_Day;
      Fecha_y_hora : Date_And_Time;
      troceado AT Fecha_y_hora : Struct
         año : Byte;
         mes : Byte;
         dia : Byte;
         hora : Byte;
         minuto : Byte;
         segundo : Byte;
         ms : Byte;
         "ms2+d_sem" : Byte;
      END_STRUCT;
      retval : Int;
      hora_convertida : ULInt;
      hora_total_string : String[9];
      hora_int : ULInt;
      minuto_int : ULInt;
      segundo_int : ULInt;
      milisegundo_int : ULInt;
   END_VAR
   VAR_TEMP   // added for the SCL form of the ladder/FBD networks
      _w1 : Bool;
   END_VAR
BEGIN

REGION Network 1: Marca que siempre esta a ON
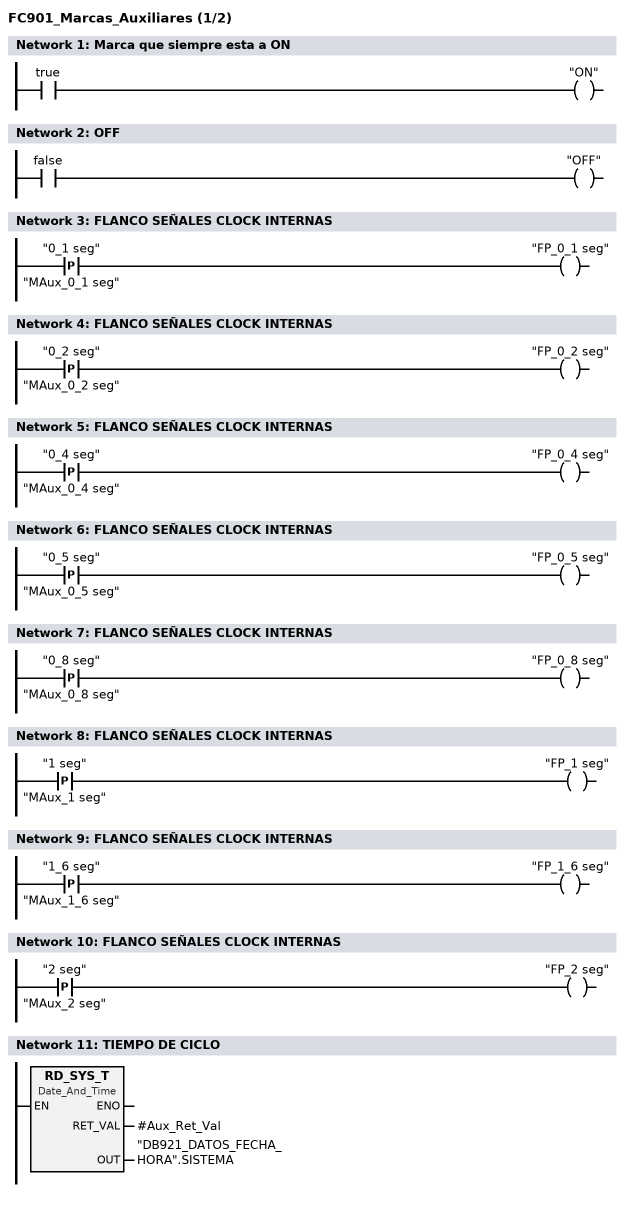
   RUNG wire#powerrail
      Contact( true )
      Coil( "ON" )
   END_RUNG
   // the same network as SCL:
   "ON" := true;
END_REGION

REGION Network 2: OFF
   RUNG wire#powerrail
      Contact( false )
      Coil( "OFF" )
   END_RUNG
   // the same network as SCL:
   "OFF" := false;
END_REGION

REGION Network 3: FLANCO SEÑALES CLOCK INTERNAS
   RUNG wire#powerrail
      P_Contact(operand := "0_1 seg", bit := "MAux_0_1 seg")
      Coil( "FP_0_1 seg" )
   END_RUNG
   // the same network as SCL:
   #_w1 := "0_1 seg" AND NOT "MAux_0_1 seg";   // rising edge of "0_1 seg"
   "MAux_0_1 seg" := "0_1 seg";
   "FP_0_1 seg" := #_w1;
END_REGION

REGION Network 4: FLANCO SEÑALES CLOCK INTERNAS
   RUNG wire#powerrail
      P_Contact(operand := "0_2 seg", bit := "MAux_0_2 seg")
      Coil( "FP_0_2 seg" )
   END_RUNG
   // the same network as SCL:
   #_w1 := "0_2 seg" AND NOT "MAux_0_2 seg";   // rising edge of "0_2 seg"
   "MAux_0_2 seg" := "0_2 seg";
   "FP_0_2 seg" := #_w1;
END_REGION

REGION Network 5: FLANCO SEÑALES CLOCK INTERNAS
   RUNG wire#powerrail
      P_Contact(operand := "0_4 seg", bit := "MAux_0_4 seg")
      Coil( "FP_0_4 seg" )
   END_RUNG
   // the same network as SCL:
   #_w1 := "0_4 seg" AND NOT "MAux_0_4 seg";   // rising edge of "0_4 seg"
   "MAux_0_4 seg" := "0_4 seg";
   "FP_0_4 seg" := #_w1;
END_REGION

REGION Network 6: FLANCO SEÑALES CLOCK INTERNAS
   RUNG wire#powerrail
      P_Contact(operand := "0_5 seg", bit := "MAux_0_5 seg")
      Coil( "FP_0_5 seg" )
   END_RUNG
   // the same network as SCL:
   #_w1 := "0_5 seg" AND NOT "MAux_0_5 seg";   // rising edge of "0_5 seg"
   "MAux_0_5 seg" := "0_5 seg";
   "FP_0_5 seg" := #_w1;
END_REGION

REGION Network 7: FLANCO SEÑALES CLOCK INTERNAS
   RUNG wire#powerrail
      P_Contact(operand := "0_8 seg", bit := "MAux_0_8 seg")
      Coil( "FP_0_8 seg" )
   END_RUNG
   // the same network as SCL:
   #_w1 := "0_8 seg" AND NOT "MAux_0_8 seg";   // rising edge of "0_8 seg"
   "MAux_0_8 seg" := "0_8 seg";
   "FP_0_8 seg" := #_w1;
END_REGION

REGION Network 8: FLANCO SEÑALES CLOCK INTERNAS
   RUNG wire#powerrail
      P_Contact(operand := "1 seg", bit := "MAux_1 seg")
      Coil( "FP_1 seg" )
   END_RUNG
   // the same network as SCL:
   #_w1 := "1 seg" AND NOT "MAux_1 seg";   // rising edge of "1 seg"
   "MAux_1 seg" := "1 seg";
   "FP_1 seg" := #_w1;
END_REGION

REGION Network 9: FLANCO SEÑALES CLOCK INTERNAS
   RUNG wire#powerrail
      P_Contact(operand := "1_6 seg", bit := "MAux_1_6 seg")
      Coil( "FP_1_6 seg" )
   END_RUNG
   // the same network as SCL:
   #_w1 := "1_6 seg" AND NOT "MAux_1_6 seg";   // rising edge of "1_6 seg"
   "MAux_1_6 seg" := "1_6 seg";
   "FP_1_6 seg" := #_w1;
END_REGION

REGION Network 10: FLANCO SEÑALES CLOCK INTERNAS
   RUNG wire#powerrail
      P_Contact(operand := "2 seg", bit := "MAux_2 seg")
      Coil( "FP_2 seg" )
   END_RUNG
   // the same network as SCL:
   #_w1 := "2 seg" AND NOT "MAux_2 seg";   // rising edge of "2 seg"
   "MAux_2 seg" := "2 seg";
   "FP_2 seg" := #_w1;
END_REGION

REGION Network 11: TIEMPO DE CICLO
   RUNG wire#powerrail
      { S7_Templates := "date_type := Date_And_Time" } RD_SYS_T(RET_VAL => #Aux_Ret_Val, OUT => "DB921_DATOS_FECHA_HORA".SISTEMA)
   END_RUNG
   // the same network as SCL:
   #Aux_Ret_Val := RD_SYS_T(OUT => "DB921_DATOS_FECHA_HORA".SISTEMA);
END_REGION

REGION Network 12
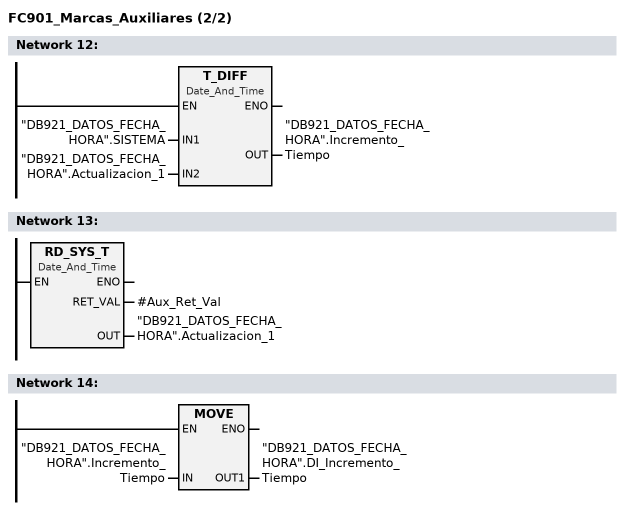
   RUNG wire#powerrail
      { S7_Templates := "[date_type := Date_And_Time, time_type := Time]" } T_DIFF(IN1 := "DB921_DATOS_FECHA_HORA".SISTEMA, IN2 := "DB921_DATOS_FECHA_HORA".Actualizacion_1, OUT => "DB921_DATOS_FECHA_HORA".Incremento_Tiempo)
   END_RUNG
   // the same network as SCL:
   T_DIFF(IN1 := "DB921_DATOS_FECHA_HORA".SISTEMA,
          IN2 := "DB921_DATOS_FECHA_HORA".Actualizacion_1,
          OUT => "DB921_DATOS_FECHA_HORA".Incremento_Tiempo);
END_REGION

REGION Network 13
   RUNG wire#powerrail
      { S7_Templates := "date_type := Date_And_Time" } RD_SYS_T(RET_VAL => #Aux_Ret_Val, OUT => "DB921_DATOS_FECHA_HORA".Actualizacion_1)
   END_RUNG
   // the same network as SCL:
   #Aux_Ret_Val := RD_SYS_T(OUT => "DB921_DATOS_FECHA_HORA".Actualizacion_1);
END_REGION

REGION Network 14
   RUNG wire#powerrail
      { S7_GenerateENO := "TRUE" } Move(in := "DB921_DATOS_FECHA_HORA".Incremento_Tiempo, out1 => "DB921_DATOS_FECHA_HORA".DI_Incremento_Tiempo)
   END_RUNG
   // the same network as SCL:
   "DB921_DATOS_FECHA_HORA".DI_Incremento_Tiempo := "DB921_DATOS_FECHA_HORA".Incremento_Tiempo;
END_REGION

REGION Network 15 (SCL)
   // GENERAR EL SELLO DE TIEMPO PARA LOS MENSAJES
   // 
   IF  "con_sello_tiempo" = true THEN

       REGION formatear_hora

           #retval := RD_LOC_T(#Fecha_y_hora);
           #hora_int := BCD16_TO_INT(#troceado.hora);
           #minuto_int := BCD16_TO_INT(#troceado.minuto);
           #segundo_int := BCD16_TO_INT(#troceado.segundo);
           #milisegundo_int := BCD16_TO_INT(#troceado.ms);
           #hora_convertida := 0;

           #hora_convertida := (#hora_int * 10000000) + (#minuto_int * 100000) + (#segundo_int * 1000) + #milisegundo_int;
           #hora_total_string := DELETE(IN := (ULINT_TO_STRING(IN := #hora_convertida)), L := 1, P := 1);

           "DB921_DATOS_FECHA_HORA".TIME_STAMP := CONCAT(IN1 := '[TIME]', IN2 := #hora_total_string);

       END_REGION

   ELSE
       "DB921_DATOS_FECHA_HORA".TIME_STAMP := '';
   END_IF;
END_REGION
END_FUNCTION

FUNCTION "FC5_Tratar_Pantalla" : Void   // FC5, LAD
{ S7_Optimized_Access := 'FALSE' }
AUTHOR : PANTALLA
NAME : 20160413
VERSION : 3.3
// stored: AutoNumber false, SetENOAutomatically false
BEGIN

REGION Network 1: Que PLC es? CCPIF A o CCPIF B o CCPIF C
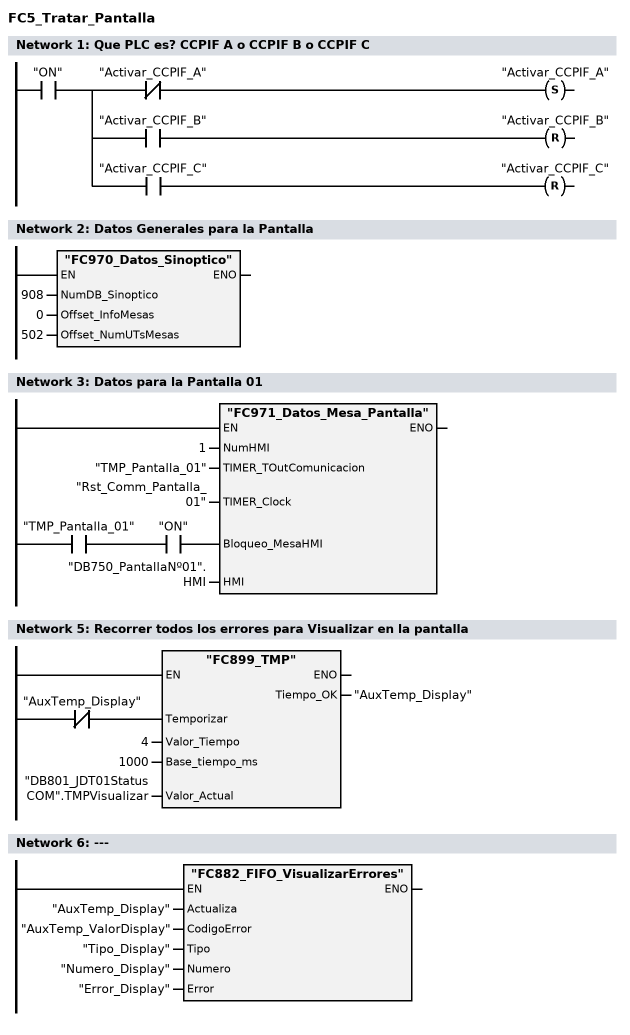
   RUNG wire#powerrail
      Contact( "ON" )
      wire#w1
      I_Contact( "Activar_CCPIF_A" )
      S_Coil( "Activar_CCPIF_A" )
   END_RUNG
   RUNG wire#w1
      Contact( "Activar_CCPIF_B" )
      R_Coil( "Activar_CCPIF_B" )
   END_RUNG
   RUNG wire#w1
      Contact( "Activar_CCPIF_C" )
      R_Coil( "Activar_CCPIF_C" )
   END_RUNG
   // the same network as SCL:
   IF "ON" AND NOT "Activar_CCPIF_A" THEN "Activar_CCPIF_A" := TRUE; END_IF;
   IF "ON" AND "Activar_CCPIF_B" THEN "Activar_CCPIF_B" := FALSE; END_IF;
   IF "ON" AND "Activar_CCPIF_C" THEN "Activar_CCPIF_C" := FALSE; END_IF;
END_REGION

REGION Network 2: Datos Generales para la Pantalla
   RUNG wire#powerrail
      "FC970_Datos_Sinoptico"(NumDB_Sinoptico := 908, Offset_InfoMesas := 0, Offset_NumUTsMesas := 502)
   END_RUNG
   // the same network as SCL:
   "FC970_Datos_Sinoptico"(NumDB_Sinoptico := 908, Offset_InfoMesas := 0, Offset_NumUTsMesas := 502);
END_REGION

REGION Network 3: Datos para la Pantalla 01
   RUNG wire#powerrail
      "FC971_Datos_Mesa_Pantalla"(Bloqueo_MesaHMI := wire#w1, NumHMI := 1, TIMER_TOutComunicacion := "TMP_Pantalla_01", TIMER_Clock := "Rst_Comm_Pantalla_01", HMI := "DB750_PantallaNº01".HMI)
   END_RUNG
   RUNG wire#powerrail
      Contact( "TMP_Pantalla_01" )
      Contact( "ON" )
   END_RUNG wire#w1
   // the same network as SCL:
   "FC971_Datos_Mesa_Pantalla"(NumHMI := 1,
                           TIMER_TOutComunicacion := "TMP_Pantalla_01",
                           TIMER_Clock := "Rst_Comm_Pantalla_01",
                           Bloqueo_MesaHMI := "TMP_Pantalla_01" AND "ON",
                           HMI := "DB750_PantallaNº01".HMI);
END_REGION

REGION Network 4: ANADIR TANTAS PANTALLAS COMO EXISTAN EN EL PROYECTO
END_REGION

REGION Network 5: Recorrer todos los errores para Visualizar en la pantalla
   RUNG wire#powerrail
      "FC899_TMP"(Valor_Tiempo := 4, Base_tiempo_ms := 1000, Tiempo_OK => "AuxTemp_Display", Valor_Actual := "DB801_JDT01StatusCOM".TMPVisualizar, Temporizar := wire#w1)
   END_RUNG
   RUNG wire#powerrail
      I_Contact( "AuxTemp_Display" )
   END_RUNG wire#w1
   // the same network as SCL:
   "FC899_TMP"(Temporizar := NOT "AuxTemp_Display",
               Valor_Tiempo := 4,
               Base_tiempo_ms := 1000,
               Valor_Actual := "DB801_JDT01StatusCOM".TMPVisualizar,
               Tiempo_OK => "AuxTemp_Display");
END_REGION

REGION Network 6: ---
   RUNG wire#powerrail
      "FC882_FIFO_VisualizarErrores"(Actualiza := "AuxTemp_Display", CodigoError := "AuxTemp_ValorDisplay", Tipo := "Tipo_Display", Numero := "Numero_Display", Error := "Error_Display")
   END_RUNG
   // the same network as SCL:
   "FC882_FIFO_VisualizarErrores"(Actualiza := "AuxTemp_Display",
                           CodigoError := "AuxTemp_ValorDisplay",
                           Tipo := "Tipo_Display",
                           Numero := "Numero_Display",
                           Error := "Error_Display");
END_REGION
END_FUNCTION

FUNCTION "FC970_Datos_Sinoptico" : Void   // FC970, LAD
TITLE = Datos Generales para la Pantalla
{ S7_Optimized_Access := 'FALSE' }
AUTHOR : PANTALLA
NAME : 20180615
VERSION : 4.3
// =- Inicializar Variables
// - Transferencia del Estado del VI para la Pantallaf
// - Nieves modificado para minimizar lineas de código
// - inicialización de Variables de mesa
// stored: AutoNumber false, SetENOAutomatically false
   VAR_INPUT
      NumDB_Sinoptico : UInt;   // DB de envio estado zonas y mesas a Pantalla
      Offset_InfoMesas : UInt;   // Byte Inicio zona de Informacion de Mesas a Pantalla
      Offset_NumUTsMesas : UInt;   // Byte Inicio zona de Numero de UTs en Mesa para Pantalla
   END_VAR
   VAR_TEMP
      ByteMesa : Struct
         Vacia : Bool;
         Cargada : Bool;
         En_Descarga : Bool;
         En_Carga : Bool;
         Etapas_Reset : Bool;
         Paro : Bool;
         Manual : Bool;
         En_Error : Bool;
      END_STRUCT;
      P_ByteMesa : DWord;
      P_Temporal : DWord;
      CNT_NumMesa : UInt;
      DB_Sinoptico : Word;
      NumeroUTs : UInt;
      NumeroUT : UInt;
      Tmp_Estado_Mesa : "EstadosMesa";
      Tmp_Estado_Maquina : "EstadoMaquina";
   END_VAR
BEGIN

NETWORK
TITLE = Inicializar Variables
// ------------------------------------------------------------------------
// --- Inicializar Variabes

      L     #NumDB_Sinoptico;  // DB Estado Zona
      T     #DB_Sinoptico;

      L     0;  // Iniciamos el contador de Mesas
      T     #CNT_NumMesa;


NETWORK
TITLE = Transferencia del Estado del VI para la Pantalla
// ------------------------------------------------------------------------
// --- Recogo el estado del VI (Mesa

BFIF: NOP   0;
// ------------------------------------------------------------------
// ---- Recoger las variables que se necesitan

      L     P##ByteMesa;  // Inicializar
      T     #P_ByteMesa;
      L     0;
      T     LB [#P_ByteMesa];

// pasamos a evaluar el estado de la mesa
// ---- 1º - Si Esta en Error
      SET;
      A     "DB900_Estado_Mesas".EstadoVI[#CNT_NumMesa].Error_Mx;
      O     "DB904_Estado_Maquinas".EstadoVI[#CNT_NumMesa].Error_MAQx;
      =     #ByteMesa.En_Error;  // Mesa En Error

// --- Si la mesa está en modo mantenimiento. NIEVES MANTENIMIENTO
      SET;
      A     "DB902_Estado_ZonaMesa".EstadoMesas[#CNT_NumMesa].Mantenimiento_CBx;
      =     #ByteMesa.Manual;
      =     #ByteMesa.Paro;
      JC    nxt;

// FIN NIEVES MANTENIMIENTO

// ---- 3º - Si Esta en Manual
      SET;
      A     "DB900_Estado_Mesas".EstadoVI[#CNT_NumMesa].Manual;
      =     #ByteMesa.Manual;
      JC    nxt;  // si está en manual no puede estar en paro

// ---- 4º - Si Esta en Paro
      SET;
      A     "DB902_Estado_ZonaMesa".EstadoMesas[#CNT_NumMesa].Paro_CBx;
      AN    #ByteMesa.Manual;  // Mesa no esta en Manual
      =     #ByteMesa.Paro;


// ---- 2º - Si Esta en Reset
// NIEVES, CAMBIO EL ORDEN PORQUE SI ESTÁ EN RESET NO ES NECESARIO SEGUIR EVALUANDO MÁS CONDICIONES

nxt:  SET;
      A     "DB900_Estado_Mesas".EstadoVI[#CNT_NumMesa].Etapas_Reset;
      =     #ByteMesa.Etapas_Reset;  // Mesa Reset
      JC    nxt2;  // salta directamente a guardar el estado en el db
// ---- 5º - Si Esta en Vacia

      SET;
      A     "DB900_Estado_Mesas".EstadoVI[#CNT_NumMesa].Etapa_Vacia;
      =     #ByteMesa.Vacia;  // Mesa Vacia
      JC    nxt2;  // si está vacía no puede estar ni cargada ni en carga ni en descarga

// ---- 6º - Si Esta en Cargada
      SET;
      A     "DB900_Estado_Mesas".EstadoVI[#CNT_NumMesa].Etapa_Cargada;
      =     #ByteMesa.Cargada;  // Mesa Cargada, no puede estar ni en carga ni en descarga
      JC    nxt2;

// ---- 7º - Si Esta en Descarga
      SET;
      A     "DB900_Estado_Mesas".EstadoVI[#CNT_NumMesa].Etapas_Descarga_S0;
      O     "DB900_Estado_Mesas".EstadoVI[#CNT_NumMesa].Etapas_Descarga_S1;
      O     "DB900_Estado_Mesas".EstadoVI[#CNT_NumMesa].Etapas_Descarga_S2;
      O     "DB900_Estado_Mesas".EstadoVI[#CNT_NumMesa].Etapas_Descarga_S3;
      O     "DB900_Estado_Mesas".EstadoVI[#CNT_NumMesa].Etapas_Descarga_S4;
      =     #ByteMesa.En_Descarga;  // Mesa En Descarga evaluamos la carga por si está en simultaneo
      JC    nxt2;

// ---- 8º - Si Esta en Carga
      SET;
      A     "DB900_Estado_Mesas".EstadoVI[#CNT_NumMesa].Etapas_Carga_E0;
      O     "DB900_Estado_Mesas".EstadoVI[#CNT_NumMesa].Etapas_Carga_E1;
      O     "DB900_Estado_Mesas".EstadoVI[#CNT_NumMesa].Etapas_Carga_E2;
      O     "DB900_Estado_Mesas".EstadoVI[#CNT_NumMesa].Etapas_Carga_E3;
      O     "DB900_Estado_Mesas".EstadoVI[#CNT_NumMesa].Etapas_Carga_E4;
      =     #ByteMesa.En_Carga;  // Mesa En Carga
      JC    nxt2;

// ------------------------------------------------------------------------
// --- Cargo el Estado del VI (Mesa) en DB Sinoptico

nxt2: L     #CNT_NumMesa;  // Puntero Origen de Datos
      L     #Offset_InfoMesas;
      +D;
      SLD   3;
      T     #P_Temporal;

      OPN   DB [#DB_Sinoptico];  // Abrir DB Destino
      L     LB [#P_ByteMesa];  // Pasarselo
      T     DBB [#P_Temporal];



NETWORK
TITLE = Calculo y Transferencia del numero de UTs en una mesa para la Pantalla
// ------------------------------------------------------------------------
// --- Calculo de la cantidad de UT's por mesa
// ----------------------------------------------------------------------------

      CALL  "FC871_NumUTsEnMesa"
      ( Mesa   := #CNT_NumMesa,
        NumUTs := #NumeroUTs
      );

// ------------------------------------------------------------------------
// --- Cargo el numero de UT's en el DB Sinoptico

      L     #CNT_NumMesa;  // Puntero Origen de Datos
      L     #Offset_NumUTsMesas;
      +D;
      SLD   3;
      T     #P_Temporal;

      OPN   DB [#DB_Sinoptico];  // Abrir DB Destino

      L     #NumeroUTs;  // Pasarselo
      T     DBB [#P_Temporal];



NETWORK
TITLE = pasar a la siguiente mesa
// ------------------------------------------------------------------------
// ------------------------------------------------------------------------
// ------------------------------------------------------------------------
// --- Pasar a la Siguiente Mesa

      L     #CNT_NumMesa;
      L     "CTE_MaxMesas";  // Si no quedan Mesas ?
      >=I;
      JC    _END;

      L     1;  //Incrementa el contador de posicion
      L     #CNT_NumMesa;
      +I;
      T     #CNT_NumMesa;

      JU    BFIF;

// ------------------------------------------------------------------------
// --- Final de la Funcion

_END: NOP   0;


END_FUNCTION

FUNCTION "FC871_NumUTsEnMesa" : Void   // FC871, LAD
{ S7_Optimized_Access := 'FALSE' }
VERSION : 1.0
// stored: AutoNumber false, SetENOAutomatically false
   VAR_INPUT
      Mesa : UInt;
   END_VAR
   VAR_OUTPUT
      NumUTs : UInt;
   END_VAR
   VAR_TEMP
      NumeroUT : UInt;
      AuxNumUTsEnMesa : UInt;
      Relleno : Byte;
      ValorReturn : Int;
   END_VAR
BEGIN

NETWORK
TITLE = ---
////////////////////////////////////////////////////////////////////////////
// --- Reseteo Variable de Salida

      L     0;
      T     #AuxNumUTsEnMesa;  // NumUTs = 0



NETWORK
TITLE = --
////////////////////////////////////////////////////////////////////////////
// --- Comprobacion de que la Mesa tenga UT o No


      L     "DB810_ColasMesas".Colas[#Mesa].UT_PrimeraMesa;
      T     #NumeroUT;

InicioBucleMesa:NOP   0;
      L     #NumeroUT;
      L     0;
      ==I;
      JC    Final;  // No hay UT's ?

      L     1;  // Incrementa el Numero de UTs en la Mesa
      L     #AuxNumUTsEnMesa;
      +I;
      T     #AuxNumUTsEnMesa;

      L     "DB812_UTs_Control".UT[#NumeroUT].UT_SiguienteMesa;
      T     #NumeroUT;

      JU    InicioBucleMesa;



NETWORK
TITLE = ---
// ----------------------------------------------------------------------------
// --- Final de la Funcion

Final:NOP   0;  // Finalizar Funcion
      L     #AuxNumUTsEnMesa;
      T     #NumUTs;


END_FUNCTION

FUNCTION "FC800_JDT01ControlTracking" : Void   // FC800, LAD
{ S7_Optimized_Access := 'FALSE' }
AUTHOR : TRACKING
NAME : 20141014
VERSION : 4.0
// stored: AutoNumber false, SetENOAutomatically false
BEGIN

NETWORK
TITLE = Previo
// -----------------------------------------------------------------------
// --- Inicialializacion
// --- Borrado de la Base de Datos

      CALL  "FC801_JDT01ControlCOM";  // Control del Puerto
      CALL  "FC806_JDT01Borrado";



NETWORK
TITLE = Distribucion Dependiendo del Tipo de JDT
///////////////////////////////////////////////////////////////////////////
///////////////////////////////////////////////////////////////////////////
///////////////////////////////////////////////////////////////////////////
/// --- Distribucion Dependiendo del Tipo de JDT (ACTUAL o VIEJO)
      SET;
      A     "Activar_JdTAntiguo";
      JC    Agencia_TrackingViejo;
      JU    Agencia_TrackingActual;



NETWORK
TITLE = Control del Sistema >>> Agencia de TRACKING ACTUAL
///////////////////////////////////////////////////////////////////////////
///////////////////////////////////////////////////////////////////////////
///////////////////////////////////////////////////////////////////////////
/// --- Agencia de TRACKING ACTUAL
Agencia_TrackingActual:NOP   0;

// ---------------------------------------------------------------------
// --- Control de Recepcion de Eventos

      CALL  "FC802_JDT01RecJdTMensaje";
      CALL  "FC804_JDT01AnalisisRecibidos";
      CALL  "FC810_EventosRecibidos"
      ( NumJDT := 1
      );

      CALL  "FC823_OrdenesMesas";
      CALL  "FC821_OrdenesDispositivos";

// ---------------------------------------------------------------------
// --- Control de EmisionEventos de Eventos


      CALL  "FC811_EventosGenerados"
      ( NumJdT := 1
      );
      CALL  "FC805_JDT01AnalisisEnviados";
      CALL  "FC803_JDT01EmiJdTMensaje";

      CALL  "FC822_EstadosMesas";
      CALL  "FC820_EstadosDispositivos";


// ---------------------------------------------------------------------
// --- Control de EmisionEventos de Router
//     *  Proceso Inicialización bucle
//     *  Eventos de la Pantalla (Movimientos)
//     *  Eventos de Reset V2.0   >>> 2023 01 05

//      CALL  "FC816_EventosEnv_Router"
//         NumJDT :=1


// NIEVES 10/04/25
      CALL  "FC717_Emision_Routing"
      ( NumJDT := 1
      );

      CALL  "FC815_EventosEnv_Control"
      ( NumJDT := 1
      );
      CALL  "FC817_EventosEnv_Reset"
      ( NumJDT := 1
      );


///////////////////////////////////////////////////////////////////////////
      JU    Fin;



NETWORK
TITLE = Control del Sistema >>> Agencia de TRACKING VIEJO
///////////////////////////////////////////////////////////////////////////
///////////////////////////////////////////////////////////////////////////
///////////////////////////////////////////////////////////////////////////
/// --- Agencia de TRACKING ACTUAL
Agencia_TrackingViejo:NOP   0;

///////////////////////////////////////////////////////////////////////////
// --- Control de Recepcion de Eventos

      CALL  "FC821_OrdenesDispositivos";


///////////////////////////////////////////////////////////////////////////
// --- Control de EmisionEventos de Eventos

      CALL  "FC811_EventosGenerados"
      ( NumJdT := 1
      );
      CALL  "FC805_JDT01AnalisisEnviados";

      CALL  "FC820_EstadosDispositivos";


///////////////////////////////////////////////////////////////////////////
      JU    Fin;



NETWORK
TITLE = Final de la Funcion
///////////////////////////////////////////////////////////////////////////
///////////////////////////////////////////////////////////////////////////
///////////////////////////////////////////////////////////////////////////
/// --- Final de la Funcion
Fin:  NOP   0;


END_FUNCTION

FUNCTION "FC810_EventosRecibidos" : Void   // FC810, LAD
TITLE = "Eventos Recibidos" - Tratamiento de los Eventos
{ S7_Optimized_Access := 'FALSE' }
AUTHOR : TRACKING
NAME : 20170707
VERSION : 4.5
// stored: AutoNumber false, SetENOAutomatically false
   VAR_INPUT
      NumJDT : UInt;
   END_VAR
   VAR_TEMP
      AtributosDeUTs : Struct   // Atributos Recibidos de las UTs
         Ruta : Array[0..20] of UInt;   // Ruta Recibida
         Etiqueta : Array[0..42] of Char;   // Etiqueta
         QUBIQA_PID : Array[0..20] of Char;   // QUBIQA - PID del Bulto
         CambiarUTDeMesa : Struct
            Origen : UInt;
            Destino : UInt;
            NOK : Bool;
            OK : Bool;
            Inicio : Bool;
            Final : Bool;
         END_STRUCT;
         AtributosTipoDeCarga : Struct
            Vacia : Bool;
            Pila : Bool;
            Remontada : Bool;
         END_STRUCT;
         Mckey : UDInt;   // Mckey
         MesaActual : UInt;   // Mesa Actual
         MesaDestino : UInt;   // Mesa Destino
         MesaIntermedia : UInt;   // Mesa Intermedia
         OrdenSalida : UInt;   // Orden de Salida
         TipoCarga : USInt;   // **** Tipo de la Carga
         Grupo : UInt;   // Grupo
         CantidadGrupo : USInt;   // Cantidad del Grupo
         PosicionGrupo : USInt;   // Posicion del Grupo
         CodigoFlejado : USInt;   // Codigo de Flejado
         CodigoEnfardado : USInt;   // Codigo de Enfradado
         CodigoEtiquetado : USInt;   // Codigo de Etiquetado
         GaliboAltura : USInt;   // Galibo - Codigo de Altura
         GaliboAnchura : USInt;   // Galibo - Codigo de Anchura
         GaliboProfundidad : USInt;   // Galibo - Codigo de Profundidad
         GaliboTaco : USInt;   // Galibo - Codigo de Taco
         GaliboHueco : USInt;   // Galibo - Codigo de Hueco
         GaliboHuecoRemontada : USInt;   // Galibo - Codigo de Hueco de Carga Remontada
         GaliboColor : USInt;   // Galibo - Codigo de Color de la Carga
         GaliboPatin : USInt;   // Galibo - Codigo de Patin
         GaliboSGA : USInt;   // Galibo - Codigo de SGA
         Presion : UInt;   // Presion de DesPaletizado o Paletizaado de Cajas de Plastico
         CotaAmarre : UInt;   // Cota de Amarre de Cajas de Plastico
         CotaAltura : UInt;   // Cota de la Altura
         CotaAnchura : UInt;   // Cota de la Anchura
         CotaProfundidad : UInt;   // Cota de la Profundidad
         Peso : UDInt;   // Peso
         PosicionDeLaEtiqueta : UInt;   // Posicion Actual de la Etiqueta
         QUBIQA_NumeroBulto : UInt;   // QUBIQA - Numero de Bulto
         QUBIQA_TotalBultos : UInt;   // QUBIQA - Numero Total de Bultos
      END_STRUCT;
      AtributosDeDispositivos : Struct   // Atributos Recibidos del Dispositivo
         TextoRecibido : Array[0..50] of Char;
         MotivoDelError : Array[0..50] of Char;   // TEXTO - Motivo del Error
         BalizaColor : "UDT_DatosBaliza";
         Tipo : UInt;   // Tipo
         Numero : UInt;   // Numero
         NuevoEstado : UInt;   // NuevoEstado
         Habilitado : UInt;
         Prioridad : UInt;
         Operacion : UInt;
         MesaHorquilla : UInt;
         MesaCargaDesCarga : UInt;
      END_STRUCT;
      VarTempUTs : Struct
         Mckey : UDInt;
         MesaActual : UInt;
         NumeroUT : UInt;
         SalidaEventoRETI : UInt;
      END_STRUCT;
      VarTempDispositivos : Struct
         Baliza : "UDT_DatosBaliza";
         Numero : UInt;
      END_STRUCT;
      DBEventosRec : Word;   // DB de Eventos Recibidos
      P_Eventos : DWord;   // Puntero al DB de Eventos Recibidos
      Evento : DWord;   // Etiqueta - Evento
      Atributo : DWord;   // Etiqueta - Atributo
      EtiquetaAtributo : DWord;   // Etiqueta - Conversion de Atributo
      NumeroEvento : UInt;   // Numero de Evento
      NumeroAtributo : UInt;   // Numero de Atributo
      Leido : UInt;
      ValorDeAtributo : UDInt;   // Valor del Atributo
      ValorDeEtiqueta : UInt;   // Valor de la Etiqueta - Conversion de Atributo
      Indice : UInt;   // Indice en el recorrido de los ARRAYs
      IndiceCBOX : UInt;
      IndiceVTDC : UInt;
      IndiceMesa : UInt;
      IndiceMaquina : UInt;
      IndiceDispositivosVarios : UInt;
      OffsetInicial : UInt;
      LonguitudTextoRecibido : UInt;
      ReturnValor : Int;
      Cero : Byte;
      JDT02_Activo : Bool;
      MesaDeJDT02 : Bool;
      DispositivoDeJDT02 : Bool;
   END_VAR
BEGIN

NETWORK
TITLE = Inicializar
/////////////////////////////////////////////////////////////////////////
/// --- Comprobar que JDT

      SET;
      R     #JDT02_Activo;
      L     "JDT1_NDB_EventosRec";  // Cogemos el DB de Eventos Recibidos
      T     #DBEventosRec;

/////////////////////////////////////////////////////////////////////////

      L     #NumJDT;
      L     2;
      <>I;
      JC    NoJdT02;

/////////////////////////////////////////////////////////////////////////

      SET;
      S     #JDT02_Activo;
      L     "JDT2_NDB_EventosRec";  // Cogemos el DB de Eventos Recibidos
      T     #DBEventosRec;

NoJdT02:NOP   0;

/////////////////////////////////////////////////////////////////////////



NETWORK
TITLE = Analizar la lista de Eventos
/////////////////////////////////////////////////////////////////////////
// Inicializar el Puntero de la Lista de Eventos

      L     0;  // Inicializar el Puntero de Eventos
      LAR2;

      OPN   DB [#DBEventosRec];  // Mirar si tiene algo el DB de Eventos Recibidos
      L     DBB [AR2, P#0.0];
      L     0;
      ==I;
      JC    NoLimpiarNada;


/////////////////////////////////////////////////////////////////////////
InicioBucle_EventosRecibidos:NOP   0;
      OPN   DB [#DBEventosRec];  // Leer el digito de Eventos Recibidos
      L     DBB [AR2, P#0.0];
      T     #Leido;

// Buscando Principio de Evento

      L     #Leido;
      L     '{';  // Inicio de Evento - '{'
      ==I;
      JC    EventosRecibidos;  // Tratar el Nuevo Evento

// Buscando el Final de la Lista de Eventos

      L     #Leido;
      L     3;  // Final de la Lista de Eventos - 0x03
      ==I;
      JC    FinalizarFuncion;  // Finalizar, ya no hay más Eventos
      L     #Leido;
      L     0;  // Final de la Lista de Eventos - 0x00 - No hay Mas
      ==I;
      JC    FinalizarFuncion;  // Finalizar, ya no hay más Eventos


/////////////////////////////////////////////////////////////////////////
FinBucle_EventosRecibidos:NOP   0;
      +AR2  P#1.0;  // Seguir recorriendo la Lista de Eventos
      JU    InicioBucle_EventosRecibidos;



NETWORK
TITLE = Distribucion de los Eventos (LIsta del DB de Conversion)
EventosRecibidos:NOP   0;

/////////////////////////////////////////////////////////////////////////
/////////////////////////////////////////////////////////////////////////
/////////////////////////////////////////////////////////////////////////
// Hay que recoger el Evento, para despues repartir
// Despues '{' va el tipo de eventos (2 Bytes)

      +AR2  P#1.0;
      OPN   DB [#DBEventosRec];
      L     DBD [AR2, P#0.0];  // Recogo el tipo de Evento (4 Caracteres)
      T     #Evento;


/////////////////////////////////////////////////////////////////////////
/////////////////////////////////////////////////////////////////////////
/////////////////////////////////////////////////////////////////////////
// Buscar numero de evento
      L     1;
      T     #NumeroEvento;
BucleDeBusqueda_NumeroDeEvento:NOP   0;

// -- Se ha encontrado el Evento Recibido
      L     "DB870_ConversorEventos".EventosRecibidos[#NumeroEvento];
      L     #Evento;
      ==D;
      JC    Encontrado_NumeroDeEvento;

// -- Final de la lista de Eventos Recibidos - No Encontrado
      L     "DB870_ConversorEventos".EventosRecibidos[#NumeroEvento];
      L     0;
      ==D;
      JC    InicioBucle_EventosRecibidos;

// --- Maximo del Array de la Lista de Eventos Recibidos - No Encontrado
      L     #NumeroEvento;
      L     "CTE_MaxArrayConversion";
      >=I;
      JC    InicioBucle_EventosRecibidos;

// --- Continuar la Busqueda
      L     #NumeroEvento;
      L     1;
      +I;
      T     #NumeroEvento;
      JU    BucleDeBusqueda_NumeroDeEvento;



NETWORK
TITLE = ----
/////////////////////////////////////////////////////////////////////////
/////////////////////////////////////////////////////////////////////////
/////////////////////////////////////////////////////////////////////////
// Distribuir dependiendo del Resultado de la Busqueda del Evento Recibido
// Para recoger los Atributos
Encontrado_NumeroDeEvento:NOP   0;
      L     #NumeroEvento;
      JL    NoExiste_NumeroDeEvento;

      JU    NoExiste_NumeroDeEvento;
      JU    Atributos_EventosDeLasUTs;  // Evento (01) - CREA
      JU    Atributos_EventosDeLasUTs;  // Evento (02) - RUTA
      JU    Atributos_EventosDeLasUTs;  // Evento (03) - DRUT
      JU    Atributos_EventosDeLasUTs;  // Evento (04) - RETI
      JU    Atributos_EventosDeLasUTs;  // Evento (05) - BORR
      JU    Atributos_EventosDeLasUTs;  // Evento (06) - DATA
      JU    Atributos_EventosDeLasUTs;  // Evento (07) - ?UT?
      JU    Atributos_EventosDeLasUTs;  // Evento (08) - MOVE
      JU    Atributos_EventosDeLasUTs;  // Evento (09) - DEMB

      JU    Atributos_EventosDeLosDispositivos;  // Evento (10) - CSTA
      JU    Atributos_EventosDeLosDispositivos;  // Evento (11) - DIDO

      JU    EventosRecibidos_Router;  // Evento (12) - ORDE
      JU    EventosRecibidos_Router;  // Evento (13) - BOET
      JU    EventosRecibidos_Router;  // Evento (14) - BOBD
      JU    EventosRecibidos_Router;  // Evento (15) - RUET
      JU    EventosRecibidos_Router;  // Evento (16) - RUES
      JU    EventosRecibidos_Router;  // Evento (17) - INIR

      JU    Atributos_EventosDeLosDispositivos;  // Evento (18) - ?ST?

      JU    EventosRecibidos_Quimarox;  // Evento (19) - QCRE
      JU    EventosRecibidos_Quimarox;  // Evento (20) - QPR?

      JU    EventosRecibidos_Reset_V2;  // Evento (21) - CHEQ

/////////////////////////////////////////////////////////////////////////
NoExiste_NumeroDeEvento:NOP   0;
      JU    InicioBucle_EventosRecibidos;



NETWORK
TITLE = Analizar la lista de los Atributos de las UTs
Atributos_EventosDeLasUTs:NOP   0;

/////////////////////////////////////////////////////////////////////////
/////////////////////////////////////////////////////////////////////////
/////////////////////////////////////////////////////////////////////////
// Inicializa variables de los Atributos de las UTs
      L     0;
      T     #Cero;

      CALL  FILL
      ( BVAL    := #Cero,
        RET_VAL := #ReturnValor,
        BLK     := #AtributosDeUTs
      );  // Inicializa Atributos de las UTS



NETWORK
TITLE = ----
/////////////////////////////////////////////////////////////////////////
/////////////////////////////////////////////////////////////////////////
// Buscando Atributos o Final del Evento
      +AR2  P#4.0;  // Prepara Puntero para ver los atributos

InicioBucleAtributos_EventosDeLasUTs:NOP   0;
      OPN   DB [#DBEventosRec];
      L     DBB [AR2, P#0.0];
      T     #Leido;

// Inicio de atributo - Ir a tratar los atributos
      L     #Leido;
      L     '[';  // '[' - Inicio de Atributo
      ==I;  // Atributo del Evento
      JC    EncontradoAtributos_EventosDeLasUTs;

// Fin del Evento
      L     #Leido;
      L     '}';  // '}' - Fin del Evento
      ==I;  // Se acabo el evento
      JC    FinalAtributos_EventosDeLasUTs;

// Sin Mensaje
      L     #Leido;
      L     0;  // No hay mas Mensaje
      ==I;  // Se acabo el evento
      JC    FinalAtributos_EventosDeLasUTs;


      +AR2  P#1.0;  // Seguir buscado atributo
      JU    InicioBucleAtributos_EventosDeLasUTs;


/////////////////////////////////////////////////////////////////////////
/////////////////////////////////////////////////////////////////////////
// Se acaba el Evento - Ir a guardar datos del Evento
FinalAtributos_EventosDeLasUTs:NOP   0;
      TAR2;
      T     #P_Eventos;  // Guardo Por donde voy en la lista de eventos
      JU    GuardarDatos_EventosRecibidos;



NETWORK
TITLE = Distribucion de los Atributos de las UTs (LIsta del DB de Conversion)
EncontradoAtributos_EventosDeLasUTs:NOP   0;

/////////////////////////////////////////////////////////////////////////
/////////////////////////////////////////////////////////////////////////
/////////////////////////////////////////////////////////////////////////
/////////////////////////////////////////////////////////////////////////
// Mirar que Atributo del Evento  es ?
      +AR2  P#1.0;
      OPN   DB [#DBEventosRec];
      L     DBD [AR2, P#0.0];  // Atributo - 4 Caracteres
      T     #Atributo;

/////////////////////////////////////////////////////////////////////////
/////////////////////////////////////////////////////////////////////////
/////////////////////////////////////////////////////////////////////////
// Buscar numero de Atributo
      L     1;
      T     #NumeroAtributo;
BucleDeBusqueda_NumeroDeAtributoDeUTs:NOP   0;

// -- Se ha encontrado el Atributo Recibido
      L     "DB870_ConversorEventos".AtributosRecibidosDeUTs[#NumeroAtributo];
      L     #Atributo;
      ==D;
      JC    Encontrado_NumeroDeAtributoDeUTs;

// -- Final de la lista de Atributo Recibidos - No Encontrado
      L     "DB870_ConversorEventos".AtributosRecibidosDeUTs[#NumeroAtributo];
      L     0;
      ==D;
      JC    InicioBucleAtributos_EventosDeLasUTs;

// --- Maximo del Array de la Lista de Atributo Recibidos - No Encontrado
      L     #NumeroAtributo;
      L     "CTE_MaxArrayConversion";
      >=I;
      JC    InicioBucleAtributos_EventosDeLasUTs;


// --- Continuar la Busqueda
      L     #NumeroAtributo;
      L     1;
      +I;
      T     #NumeroAtributo;
      JU    BucleDeBusqueda_NumeroDeAtributoDeUTs;



NETWORK
TITLE = ----
/////////////////////////////////////////////////////////////////////////
/////////////////////////////////////////////////////////////////////////
/////////////////////////////////////////////////////////////////////////
// Distribuir dependiendo del Resultado de la Busqueda de Atributo Recibido
Encontrado_NumeroDeAtributoDeUTs:NOP   0;
      L     #NumeroAtributo;
      JL    NoExiste_NumeroDeAtibutoDeUTs;

      JU    NoExiste_NumeroDeAtibutoDeUTs;
      JU    AtributoDeUTs_MCKY;  // Atributo (01) - MCKY
      JU    AtributoDeUTs_MESA;  // Atributo (02) - MESA
      JU    AtributoDeUTs_RUTA;  // Atributo (03) - RUTA
      JU    AtributoDeUTs_SALI;  // Atributo (04) - SALI
      JU    AtributoDeUTs_SSCC;  // Atributo (05) - SSCC

      JU    AtributoDeUTs_GRUP;  // Atributo (06) - GRUP
      JU    AtributoDeUTs_GCNT;  // Atributo (07) - GCNT
      JU    AtributoDeUTs_GORD;  // Atributo (08) - GORD

      JU    AtributoDeUTs_FLEJ;  // Atributo (09) - FLEJ
      JU    AtributoDeUTs_ENFA;  // Atributo (10) - ENFA
      JU    AtributoDeUTs_ETIQ;  // Atributo (11) - ETIQ

      JU    AtributoDeUTs_AMAR;  // Atributo (12) - AMAR
      JU    AtributoDeUTs_PRES;  // Atributo (13) - PRES

      JU    AtributoDeUTs_NBUL_QUBIQA;  // Atributo (14) - NBUL (QUBIQA)
      JU    AtributoDeUTs_NTBU_QUBIQA;  // Atributo (15) - NTBU (QUBIQA)
      JU    AtributoDeUTs_PID_QUBIQA;  // Atributo (16) - PID_ (QUBIQA)

      JU    AtributoDeUTs_TIPO;  // Atributo (17) - TIPO
      JU    AtributoDeUTs_REMO;  // Atributo (18) - REMO
      JU    AtributoDeUTs_PILA;  // Atributo (19) - PILA
      JU    AtributoDeUTs_VACI;  // Atributo (20) - VACI

      JU    AtributoDeUTs_COTA;  // Atributo (21) - COTA
      JU    AtributoDeUTs_COTW;  // Atributo (22) - COTW
      JU    AtributoDeUTs_COTL;  // Atributo (23) - COTL
      JU    AtributoDeUTs_PESO;  // Atributo (24) - PESO

      JU    AtributoDeUTs_ALTO;  // Atributo (25) - ALTO
      JU    AtributoDeUTs_ANCH;  // Atributo (26) - ANCH
      JU    AtributoDeUTs_PROF;  // Atributo (27) - PROF
      JU    AtributoDeUTs_TACO;  // Atributo (28) - TACO
      JU    AtributoDeUTs_HUEC;  // Atributo (29) - HUEC
      JU    AtributoDeUTs_HUER;  // Atributo (30) - HUER
      JU    AtributoDeUTs_COLO;  // Atributo (31) - COLO
      JU    AtributoDeUTs_PATI;  // Atributo (32) - PATI

      JU    AtributoDeUTs_LETI;  // Atributo (33) - LETI

      JU    AtributoDeUTs_SGAP;  // Atributo (34) - SGAP
      JU    AtributoDeUTs_SGAE;  // Atributo (35) - SGAE
      JU    AtributoDeUTs_SGAD;  // Atributo (36) - SGAD
      JU    AtributoDeUTs_SGA_Error;  // Atributo (37) - SGA

      JU    AtributoDeUTs_RSLT;  // Atributo (38) - RSLT
      JU    AtributoDeUTs_PDST;  // Atributo (39) - PDST
      JU    AtributoDeUTs_DEST;  // Atributo (40) - DEST

      JU    AtributoDeUTs_FLEJ;  // Atributo (41) - PALE >>> NDD

/////////////////////////////////////////////////////////////////////////
NoExiste_NumeroDeAtibutoDeUTs:NOP   0;
      JU    InicioBucleAtributos_EventosDeLasUTs;



NETWORK
TITLE = ---- ---- Recoger el Atributo de las UTs - MCKY
/////////////////////////////////////////////////////////////////////////
/////////////////////////////////////////////////////////////////////////
/////////////////////////////////////////////////////////////////////////
AtributoDeUTs_MCKY:NOP   0;
      +AR2  P#5.0;
      TAR2;
      T     #P_Eventos;
      SRD   3;
      T     #OffsetInicial;

// Obtener el Valor del Atributo
      CALL  "FC892_Obtener_ValorDelAtributo"
      ( DB_String := #DBEventosRec,
        OffsetIni := #OffsetInicial,
        Valor     := #ValorDeAtributo
      );

      L     #ValorDeAtributo;  // Lo guardo
      T     #AtributosDeUTs.Mckey;

// Continuo con el Evento
      L     #P_Eventos;
      LAR2;
      JU    InicioBucleAtributos_EventosDeLasUTs;



NETWORK
TITLE = ---- ---- Recoger el Atributo de las UTs - MESA
/////////////////////////////////////////////////////////////////////////
/////////////////////////////////////////////////////////////////////////
/////////////////////////////////////////////////////////////////////////
AtributoDeUTs_MESA:NOP   0;
      +AR2  P#5.0;
      TAR2;
      T     #P_Eventos;
      SRD   3;
      T     #OffsetInicial;

// Obtener el Valor del Atributo
      CALL  "FC892_Obtener_ValorDelAtributo"
      ( DB_String := #DBEventosRec,
        OffsetIni := #OffsetInicial,
        Valor     := #ValorDeAtributo
      );

      L     #ValorDeAtributo;  // Lo guardo
      T     #AtributosDeUTs.MesaActual;

// Continuo con el Evento
      L     #P_Eventos;
      LAR2;
      JU    InicioBucleAtributos_EventosDeLasUTs;



NETWORK
TITLE = ---- ---- Recoger el Atributo de las UTs - RUTA
/////////////////////////////////////////////////////////////////////////
/////////////////////////////////////////////////////////////////////////
/////////////////////////////////////////////////////////////////////////
AtributoDeUTs_RUTA:NOP   0;
      +AR2  P#5.0;  // Preparo punteros
      L     0;
      T     #Indice;

/////////////////////////////////////////////////////////////////////////
// Inicio para recoger la nueva ruta
InicioBucleAtributoDeUTs_RUTA:NOP   0;
      OPN   DB [#DBEventosRec];
      L     DBB [AR2, P#0.0];
      T     #Leido;

// Mirar si es nueva mesa o final de ruta

      L     #Leido;
      L     '[';  // Nueva ruta de la Mesa
      ==I;
      JC    NuevaMesaAtributoDeUTs_RUTA;
      L     #Leido;
      L     ')';  // Es Final de Ruta
      ==I;
      JC    FinalBucleAtributoDeUTs_RUTA;

      +AR2  P#1.0;  // Continuar hasta encontrar otra Mesa de la ruta
      JU    InicioBucleAtributoDeUTs_RUTA;


/////////////////////////////////////////////////////////////////////////
// Nueva mesa para la ruta, recogerla y guradarla
NuevaMesaAtributoDeUTs_RUTA:NOP   0;
      +AR2  P#6.0;
      TAR2;
      T     #P_Eventos;
      SRD   3;
      T     #OffsetInicial;

// Obtener el Valor de la Mesa de la Ruta

      CALL  "FC892_Obtener_ValorDelAtributo"
      ( DB_String := #DBEventosRec,
        OffsetIni := #OffsetInicial,
        Valor     := #ValorDeAtributo
      );
      L     #ValorDeAtributo;  // Lo guardo
      T     #AtributosDeUTs.Ruta[#Indice];
      T     #AtributosDeUTs.MesaDestino;

      L     #Indice;  // Siguiente Mesa de la Ruta
      L     1;
      +I;
      T     #Indice;

      L     0;  //Se pone a 0 para indicar final de ruta
      T     #AtributosDeUTs.Ruta[#Indice];

      L     #P_Eventos;
      LAR2;
      JU    InicioBucleAtributoDeUTs_RUTA;


/////////////////////////////////////////////////////////////////////////
// No tiene más mesas la ruta. Continuo con el Evento
FinalBucleAtributoDeUTs_RUTA:NOP   0;
      L     #AtributosDeUTs.Ruta[0];  // Mesa Intermedia la primera mesa de la Ruta
      T     #AtributosDeUTs.MesaIntermedia;

      L     #P_Eventos;
      LAR2;
      JU    InicioBucleAtributos_EventosDeLasUTs;



NETWORK
TITLE = ---- ---- Recoger el Atributo de las UTs - SALI
/////////////////////////////////////////////////////////////////////////
/////////////////////////////////////////////////////////////////////////
/////////////////////////////////////////////////////////////////////////
AtributoDeUTs_SALI:NOP   0;
      +AR2  P#5.0;
      TAR2;
      T     #P_Eventos;
      SRD   3;
      T     #OffsetInicial;

// Obtener el Valor del Atributo
      CALL  "FC892_Obtener_ValorDelAtributo"
      ( DB_String := #DBEventosRec,
        OffsetIni := #OffsetInicial,
        Valor     := #ValorDeAtributo
      );

      L     #ValorDeAtributo;  // Lo guardo
      T     #AtributosDeUTs.OrdenSalida;

// Continuo con el Evento
      L     #P_Eventos;
      LAR2;
      JU    InicioBucleAtributos_EventosDeLasUTs;



NETWORK
TITLE = ---- ---- Recoger el Atributo de las UTs - SSCC
/////////////////////////////////////////////////////////////////////////
/////////////////////////////////////////////////////////////////////////
/////////////////////////////////////////////////////////////////////////
AtributoDeUTs_SSCC:NOP   0;
      +AR2  P#5.0;
      L     2;
      T     #Indice;

/////////////////////////////////////////////////////////////////////////
// Inicio a recoger la etiqueta
InicioBucleAtributoDeUTs_Etiqueta:NOP   0;
      OPN   DB [#DBEventosRec];
      L     DBB [AR2, P#0.0];
      T     #Leido;

      L     #Leido;
      L     '}';  // Es Final de etiqueta
      ==I;
      JC    FinalBucleAtributoDeUTs_Etiqueta;
      L     #Leido;
      L     '[';  // Es Final de etiqueta
      ==I;
      JC    FinalBucleAtributoDeUTs_Etiqueta;

      L     #Leido;
      T     #AtributosDeUTs.Etiqueta[#Indice];

      L     #Indice;  // Siguiente caracter
      L     1;
      +I;
      T     #Indice;
      +AR2  P#1.0;

      L     0;
      T     #AtributosDeUTs.Etiqueta[#Indice];
      JU    InicioBucleAtributoDeUTs_Etiqueta;

/////////////////////////////////////////////////////////////////////////
FinalBucleAtributoDeUTs_Etiqueta:NOP   0;
      L     40;  // Inicio la carcacteristica de la STRING
      T     #AtributosDeUTs.Etiqueta[0];
      L     #Indice;
      L     2;
      -I;
      T     #AtributosDeUTs.Etiqueta[1];

      JU    InicioBucleAtributos_EventosDeLasUTs;



NETWORK
TITLE = ---- ---- Recoger el Atributo de las UTs - GRUP
/////////////////////////////////////////////////////////////////////////
/////////////////////////////////////////////////////////////////////////
/////////////////////////////////////////////////////////////////////////
AtributoDeUTs_GRUP:NOP   0;
      +AR2  P#5.0;
      TAR2;
      T     #P_Eventos;
      SRD   3;
      T     #OffsetInicial;

// Obtener el Valor del Atributo
      CALL  "FC892_Obtener_ValorDelAtributo"
      ( DB_String := #DBEventosRec,
        OffsetIni := #OffsetInicial,
        Valor     := #ValorDeAtributo
      );

      L     #ValorDeAtributo;  // Lo guardo
      T     #AtributosDeUTs.Grupo;

// Continuo con el Evento
      L     #P_Eventos;
      LAR2;
      JU    InicioBucleAtributos_EventosDeLasUTs;



NETWORK
TITLE = ---- ---- Recoger el Atributo de las UTs - GCNT (Cantidad de UTs en el Grupo)
/////////////////////////////////////////////////////////////////////////
/////////////////////////////////////////////////////////////////////////
/////////////////////////////////////////////////////////////////////////
AtributoDeUTs_GCNT:NOP   0;
      +AR2  P#5.0;
      TAR2;
      T     #P_Eventos;
      SRD   3;
      T     #OffsetInicial;

// Obtener el Valor del Atributo
      CALL  "FC892_Obtener_ValorDelAtributo"
      ( DB_String := #DBEventosRec,
        OffsetIni := #OffsetInicial,
        Valor     := #ValorDeAtributo
      );

      L     #ValorDeAtributo;  // Lo guardo
      T     #AtributosDeUTs.CantidadGrupo;

// Continuo con el Evento
      L     #P_Eventos;
      LAR2;
      JU    InicioBucleAtributos_EventosDeLasUTs;



NETWORK
TITLE = ---- ---- Recoger el Atributo de las UTs - GORD (Posicion en el Grupo)
/////////////////////////////////////////////////////////////////////////
/////////////////////////////////////////////////////////////////////////
/////////////////////////////////////////////////////////////////////////
AtributoDeUTs_GORD:NOP   0;
      +AR2  P#5.0;
      TAR2;
      T     #P_Eventos;
      SRD   3;
      T     #OffsetInicial;

// Obtener el Valor del Atributo
      CALL  "FC892_Obtener_ValorDelAtributo"
      ( DB_String := #DBEventosRec,
        OffsetIni := #OffsetInicial,
        Valor     := #ValorDeAtributo
      );

      L     #ValorDeAtributo;  // Lo guardo
      T     #AtributosDeUTs.PosicionGrupo;

// Continuo con el Evento
      L     #P_Eventos;
      LAR2;
      JU    InicioBucleAtributos_EventosDeLasUTs;



NETWORK
TITLE = ---- ---- Recoger el Atributo de las UTs - FLEJ (Codigo de Flejado)
/////////////////////////////////////////////////////////////////////////
/////////////////////////////////////////////////////////////////////////
/////////////////////////////////////////////////////////////////////////
AtributoDeUTs_FLEJ:NOP   0;
      +AR2  P#5.0;
      TAR2;
      T     #P_Eventos;
      SRD   3;
      T     #OffsetInicial;

// Obtener el Valor del Atributo
      CALL  "FC892_Obtener_ValorDelAtributo"
      ( DB_String := #DBEventosRec,
        OffsetIni := #OffsetInicial,
        Valor     := #ValorDeAtributo
      );

      L     #ValorDeAtributo;  // Lo guardo
      T     #AtributosDeUTs.CodigoFlejado;

// Continuo con el Evento
      L     #P_Eventos;
      LAR2;
      JU    InicioBucleAtributos_EventosDeLasUTs;



NETWORK
TITLE = ---- ---- Recoger el Atributo de las UTs - ENFA (Codigo de Enfardado)
/////////////////////////////////////////////////////////////////////////
/////////////////////////////////////////////////////////////////////////
/////////////////////////////////////////////////////////////////////////
AtributoDeUTs_ENFA:NOP   0;
      +AR2  P#5.0;
      TAR2;
      T     #P_Eventos;
      SRD   3;
      T     #OffsetInicial;

// Obtener el Valor del Atributo
      CALL  "FC892_Obtener_ValorDelAtributo"
      ( DB_String := #DBEventosRec,
        OffsetIni := #OffsetInicial,
        Valor     := #ValorDeAtributo
      );

      L     #ValorDeAtributo;  // Lo guardo
      T     #AtributosDeUTs.CodigoEnfardado;

// Continuo con el Evento
      L     #P_Eventos;
      LAR2;
      JU    InicioBucleAtributos_EventosDeLasUTs;



NETWORK
TITLE = ---- ---- Recoger el Atributo de las UTs - ETIQ (Codigo de Etiquetado)
/////////////////////////////////////////////////////////////////////////
/////////////////////////////////////////////////////////////////////////
/////////////////////////////////////////////////////////////////////////
AtributoDeUTs_ETIQ:NOP   0;
      +AR2  P#5.0;
      TAR2;
      T     #P_Eventos;
      SRD   3;
      T     #OffsetInicial;

// Obtener el Valor del Atributo
      CALL  "FC892_Obtener_ValorDelAtributo"
      ( DB_String := #DBEventosRec,
        OffsetIni := #OffsetInicial,
        Valor     := #ValorDeAtributo
      );

      L     #ValorDeAtributo;  // Lo guardo
      T     #AtributosDeUTs.CodigoEtiquetado;

// Continuo con el Evento
      L     #P_Eventos;
      LAR2;
      JU    InicioBucleAtributos_EventosDeLasUTs;



NETWORK
TITLE = ---- ---- Recoger el Atributo de las UTs - AMAR (Cota de Amarre de las Cajas de Plastico)
/////////////////////////////////////////////////////////////////////////
/////////////////////////////////////////////////////////////////////////
/////////////////////////////////////////////////////////////////////////
AtributoDeUTs_AMAR:NOP   0;
      +AR2  P#5.0;
      TAR2;
      T     #P_Eventos;
      SRD   3;
      T     #OffsetInicial;

// Obtener el Valor del Atributo
      CALL  "FC892_Obtener_ValorDelAtributo"
      ( DB_String := #DBEventosRec,
        OffsetIni := #OffsetInicial,
        Valor     := #ValorDeAtributo
      );

      L     #ValorDeAtributo;  // Lo guardo
      T     #AtributosDeUTs.CotaAmarre;

// Continuo con el Evento
      L     #P_Eventos;
      LAR2;
      JU    InicioBucleAtributos_EventosDeLasUTs;



NETWORK
TITLE = ---- ---- Recoger el Atributo de las UTs - PRES (Presion para el Paletizador y DesPaletizador de las Cajas de Plastico) /// OJOOOOOOO
/////////////////////////////////////////////////////////////////////////
/////////////////////////////////////////////////////////////////////////
/////////////////////////////////////////////////////////////////////////
AtributoDeUTs_PRES:NOP   0;
      +AR2  P#5.0;
      TAR2;
      T     #P_Eventos;
      SRD   3;
      T     #OffsetInicial;

// Obtener el Valor del Atributo
      CALL  "FC892_Obtener_ValorDelAtributo"
      ( DB_String := #DBEventosRec,
        OffsetIni := #OffsetInicial,
        Valor     := #ValorDeAtributo
      );

      L     #ValorDeAtributo;  // Lo guardo
      T     #AtributosDeUTs.Presion;

// Continuo con el Evento
      L     #P_Eventos;
      LAR2;
      JU    InicioBucleAtributos_EventosDeLasUTs;



NETWORK
TITLE = ---- ---- Recoger el Atributo de las UTs - NBUL (QUBIQA - Nurmero de Bulto)
/////////////////////////////////////////////////////////////////////////
/////////////////////////////////////////////////////////////////////////
/////////////////////////////////////////////////////////////////////////
AtributoDeUTs_NBUL_QUBIQA:NOP   0;
      +AR2  P#5.0;
      TAR2;
      T     #P_Eventos;
      SRD   3;
      T     #OffsetInicial;

// Obtener el Valor del Atributo
      CALL  "FC892_Obtener_ValorDelAtributo"
      ( DB_String := #DBEventosRec,
        OffsetIni := #OffsetInicial,
        Valor     := #ValorDeAtributo
      );

      L     #ValorDeAtributo;  // Lo guardo
      T     #AtributosDeUTs.QUBIQA_NumeroBulto;

// Continuo con el Evento
      L     #P_Eventos;
      LAR2;
      JU    InicioBucleAtributos_EventosDeLasUTs;



NETWORK
TITLE = ---- ---- Recoger el Atributo de las UTs - NTBU (QUBIQA - Numerom Total de Bultos)
/////////////////////////////////////////////////////////////////////////
/////////////////////////////////////////////////////////////////////////
/////////////////////////////////////////////////////////////////////////
AtributoDeUTs_NTBU_QUBIQA:NOP   0;
      +AR2  P#5.0;
      TAR2;
      T     #P_Eventos;
      SRD   3;
      T     #OffsetInicial;

// Obtener el Valor del Atributo
      CALL  "FC892_Obtener_ValorDelAtributo"
      ( DB_String := #DBEventosRec,
        OffsetIni := #OffsetInicial,
        Valor     := #ValorDeAtributo
      );

      L     #ValorDeAtributo;  // Lo guardo
      T     #AtributosDeUTs.QUBIQA_TotalBultos;

// Continuo con el Evento
      L     #P_Eventos;
      LAR2;
      JU    InicioBucleAtributos_EventosDeLasUTs;



NETWORK
TITLE = ---- ---- Recoger el Atributo de las UTs - PID_ (QIBIQA - PID del Bulto - 20 Caracteres)
/////////////////////////////////////////////////////////////////////////
/////////////////////////////////////////////////////////////////////////
/////////////////////////////////////////////////////////////////////////
AtributoDeUTs_PID_QUBIQA:NOP   0;
      +AR2  P#5.0;
      L     0;
      T     #Indice;

/////////////////////////////////////////////////////////////////////////
// Inicio a recoger la etiqueta
InicioBucleAtributoDeUTs_PID_QUBIQA:NOP   0;
      OPN   DB [#DBEventosRec];
      L     DBB [AR2, P#0.0];
      T     #Leido;

      L     #Leido;
      L     '}';  // Es Final de etiqueta
      ==I;
      JC    FinalBucleAtributoDeUTs_PID_QUBIQA;
      L     #Leido;
      L     '[';  // Es Final de etiqueta
      ==I;
      JC    FinalBucleAtributoDeUTs_PID_QUBIQA;

      L     #Leido;
      T     #AtributosDeUTs.QUBIQA_PID[#Indice];

      L     #Indice;  // Siguiente caracter
      L     1;
      +I;
      T     #Indice;
      +AR2  P#1.0;

      L     0;
      T     #AtributosDeUTs.QUBIQA_PID[#Indice];
      JU    InicioBucleAtributoDeUTs_PID_QUBIQA;

/////////////////////////////////////////////////////////////////////////
FinalBucleAtributoDeUTs_PID_QUBIQA:NOP   0;
      JU    InicioBucleAtributos_EventosDeLasUTs;



NETWORK
TITLE = ---- ---- Recoger el Atributo de las UTs - TIPO (Tipo de Carga) ****
/////////////////////////////////////////////////////////////////////////
/////////////////////////////////////////////////////////////////////////
/////////////////////////////////////////////////////////////////////////
AtributoDeUTs_TIPO:NOP   0;
      +AR2  P#5.0;

      OPN   DB [#DBEventosRec];
      L     DBD [AR2, P#0.0];
      T     #EtiquetaAtributo;

// Obtener el Valor del Atributo
      CALL  "FC894_Obtener_ValorDeEtiqueta"
      ( EtiquetaEvento := #EtiquetaAtributo,
        ValorEvento    := #ValorDeEtiqueta
      );

      L     #ValorDeEtiqueta;  // Lo guardo
      T     #AtributosDeUTs.TipoCarga;


// Continuo con el Evento
      +AR2  P#4.0;
      JU    InicioBucleAtributos_EventosDeLasUTs;



NETWORK
TITLE = ---- ---- Recoger el Atributo de las UTs - REMO (La Carga esta Remontada)
/////////////////////////////////////////////////////////////////////////
/////////////////////////////////////////////////////////////////////////
/////////////////////////////////////////////////////////////////////////
AtributoDeUTs_REMO:NOP   0;
      +AR2  P#5.0;

      OPN   DB [#DBEventosRec];
      L     DBB [AR2, P#0.0];  // Sacar el Valor del Campo
      T     #Leido;
      +AR2  P#1.0;

      L     #Leido;  // Comparar si es cero
      L     '0';  // La carga No Esta Remontada ?
      ==I;
      JC    InicioBucleAtributos_EventosDeLasUTs;

      SET;
      S     #AtributosDeUTs.AtributosTipoDeCarga.Remontada;


// Continuo con el Evento
      JU    InicioBucleAtributos_EventosDeLasUTs;



